LIN {X 0,Y 246.52,Z 385.054,A -85,B 0,C 180,E1 -18943.173,E2 -18943.173} C_VEL
LIN {X 0,Y 246.538,Z 383.912,A -85,B 0,C 180,E1 -18945.451,E2 -18945.451} C_VEL
LIN {X 0,Y 246.771,Z 381.922,A -85,B 0,C 180,E1 -18947.771,E2 -18947.771} C_VEL
LIN {X 0,Y 247.108,Z 378.922,A -85,B 0,C 180,E1 -18950.165,E2 -18950.165} C_VEL
LIN {X 0,Y 247.698,Z 374.789,A -85,B 0,C 180,E1 -18952.602,E2 -18952.602} C_VEL
LIN {X 0,Y 248.557,Z 368.103,A -85,B 0,C 180,E1 -18955.564,E2 -18955.564} C_VEL
LIN {X 0,Y 249.777,Z 360.458,A -85,B 0,C 180,E1 -18958.176,E2 -18958.176} C_VEL
LIN {X 0,Y 250.952,Z 352.88,A -85,B 0,C 180,E1 -18960.245,E2 -18960.245} C_VEL
LIN {X 0,Y 252.424,Z 343.571,A -85,B 0,C 180,E1 -18962.309,E2 -18962.309} C_VEL
LIN {X 0,Y 253.973,Z 333.387,A -85,B 0,C 180,E1 -18964.133,E2 -18964.133} C_VEL
LIN {X 0,Y 255.381,Z 323.073,A -85,B 0,C 180,E1 -18965.62,E2 -18965.62} C_VEL
LIN {X 0,Y 256.697,Z 311.556,A -85,B 0,C 180,E1 -18966.931,E2 -18966.931} C_VEL
LIN {X 0,Y 257.975,Z 298.577,A -85,B 0,C 180,E1 -18968.044,E2 -18968.044} C_VEL
LIN {X 0,Y 258.876,Z 285.337,A -85,B 0,C 180,E1 -18968.84,E2 -18968.84} C_VEL
LIN {X 0,Y 259.602,Z 268.509,A -85,B 0,C 180,E1 -18969.443,E2 -18969.443} C_VEL
LIN {X 0,Y 261.737,Z 209.958,A -85,B 0,C 180,E1 -18971.254,E2 -18971.254} C_VEL
LIN {X 0,Y 260.436,Z 204.838,A -85,B 0,C 180,E1 -18971.54,E2 -18971.54} C_VEL
LIN {X 0,Y 251.175,Z 178.768,A -85,B 0,C 180,E1 -18973.282,E2 -18973.282} C_VEL
LIN {X 0,Y 249.486,Z 174.092,A -85,B 0,C 180,E1 -18973.639,E2 -18973.639} C_VEL
LIN {X 0,Y 249.178,Z 172.45,A -85,B 0,C 180,E1 -18974.354,E2 -18974.354} C_VEL
LIN {X 0,Y 249.215,Z 172.443,A -85,B 0,C 180,E1 -18978.615,E2 -18978.615} C_VEL
LIN {X 0,Y 249.411,Z 172.416,A -85,B 0,C 180,E1 -18981.901,E2 -18981.901} C_VEL
LIN {X 0,Y 249.258,Z 172.435,A -85,B 0,C 180,E1 -18985.148,E2 -18985.148} C_VEL
LIN {X 0,Y 249.654,Z 172.389,A -85,B 0,C 180,E1 -18988.387,E2 -18988.387} C_VEL
LIN {X 0,Y 249.652,Z 172.389,A -85,B 0,C 180,E1 -18991.613,E2 -18991.613} C_VEL
LIN {X 0,Y 249.424,Z 172.416,A -85,B 0,C 180,E1 -18996.472,E2 -18996.472} C_VEL
LIN {X 0,Y 249.33,Z 172.43,A -85,B 0,C 180,E1 -18999.737,E2 -18999.737} C_VEL
LIN {X 0,Y 249.143,Z 172.45,A -85,B 0,C 180,E1 -19004.707,E2 -19004.707} C_VEL
LIN {X 0,Y 249.075,Z 172.459,A -85,B 0,C 180,E1 -19008.082,E2 -19008.082} C_VEL
LIN {X 0,Y 249.039,Z 172.464,A -85,B 0,C 180,E1 -19011.522,E2 -19011.522} C_VEL
LIN {X 0,Y 249.04,Z 172.464,A -85,B 0,C 180,E1 -19015.44,E2 -19015.44} C_VEL
LIN {X 0,Y 249.02,Z 172.465,A -85,B 0,C 180,E1 -19018.968,E2 -19018.968} C_VEL
LIN {X 0,Y 249.022,Z 172.457,A -85,B 0,C 180,E1 -19022.427,E2 -19022.427} C_VEL
LIN {X 0,Y 249.023,Z 172.463,A -85,B 0,C 180,E1 -19026.346,E2 -19026.346} C_VEL
LIN {X 0,Y 248.975,Z 172.467,A -85,B 0,C 180,E1 -19030.484,E2 -19030.484} C_VEL
LIN {X 0,Y 248.958,Z 172.467,A -85,B 0,C 180,E1 -19034.889,E2 -19034.889} C_VEL
LIN {X 0,Y 248.975,Z 172.471,A -85,B 0,C 180,E1 -19037.355,E2 -19037.355} C_VEL
LIN {X 0,Y 249.036,Z 172.461,A -85,B 0,C 180,E1 -19042.202,E2 -19042.202} C_VEL
LIN {X 0,Y 249.039,Z 172.452,A -85,B 0,C 180,E1 -19045.64,E2 -19045.64} C_VEL
LIN {X 0,Y 248.998,Z 172.463,A -85,B 0,C 180,E1 -19049.467,E2 -19049.467} C_VEL
LIN {X 0,Y 249.017,Z 172.465,A -85,B 0,C 180,E1 -19053.157,E2 -19053.157} C_VEL
LIN {X 0,Y 249.002,Z 172.466,A -85,B 0,C 180,E1 -19056.726,E2 -19056.726} C_VEL
LIN {X 0,Y 249.038,Z 172.456,A -85,B 0,C 180,E1 -19060.206,E2 -19060.206} C_VEL
LIN {X 0,Y 249.155,Z 172.44,A -85,B 0,C 180,E1 -19063.617,E2 -19063.617} C_VEL
LIN {X 0,Y 249.214,Z 172.44,A -85,B 0,C 180,E1 -19068.615,E2 -19068.615} C_VEL
LIN {X 0,Y 249.399,Z 172.415,A -85,B 0,C 180,E1 -19071.901,E2 -19071.901} C_VEL
LIN {X 0,Y 249.249,Z 172.424,A -85,B 0,C 180,E1 -19075.148,E2 -19075.148} C_VEL
LIN {X 0,Y 249.651,Z 172.385,A -85,B 0,C 180,E1 -19078.388,E2 -19078.388} C_VEL
LIN {X 0,Y 249.651,Z 172.386,A -85,B 0,C 180,E1 -19081.614,E2 -19081.614} C_VEL
LIN {X 0,Y 249.383,Z 172.411,A -85,B 0,C 180,E1 -19087.292,E2 -19087.292} C_VEL
LIN {X 0,Y 249.329,Z 172.426,A -85,B 0,C 180,E1 -19089.738,E2 -19089.738} C_VEL
LIN {X 0,Y 249.128,Z 172.447,A -85,B 0,C 180,E1 -19094.277,E2 -19094.277} C_VEL
LIN {X 0,Y 248.465,Z 172.533,A -85,B 0,C 180,E1 -19095.626,E2 -19095.626} C_VEL
LIN {X 0,Y 245.549,Z 172.897,A -85,B 0,C 180,E1 -19097.823,E2 -19097.823} C_VEL
LIN {X 0,Y 243.077,Z 173.207,A -85,B 0,C 180,E1 -19099.613,E2 -19099.613} C_VEL
LIN {X 0,Y 242.044,Z 173.334,A -85,B 0,C 180,E1 -19101.004,E2 -19101.004} C_VEL
LIN {X 0,Y 241.976,Z 173.344,A -85,B 0,C 180,E1 -19101.475,E2 -19101.475} C_VEL
LIN {X 0,Y 241.985,Z 173.343,A -85,B 0,C 180,E1 -19105.827,E2 -19105.827} C_VEL
LIN {X 0,Y 241.962,Z 173.345,A -85,B 0,C 180,E1 -19109.59,E2 -19109.59} C_VEL
LIN {X 0,Y 241.978,Z 173.334,A -85,B 0,C 180,E1 -19113.494,E2 -19113.494} C_VEL
LIN {X 0,Y 241.983,Z 173.343,A -85,B 0,C 180,E1 -19117.584,E2 -19117.584} C_VEL
LIN {X 0,Y 241.908,Z 173.351,A -85,B 0,C 180,E1 -19121.93,E2 -19121.93} C_VEL
LIN {X 0,Y 241.901,Z 173.353,A -85,B 0,C 180,E1 -19126.581,E2 -19126.581} C_VEL
LIN {X 0,Y 241.993,Z 173.341,A -85,B 0,C 180,E1 -19131.642,E2 -19131.642} C_VEL
LIN {X 0,Y 242.041,Z 173.508,A -85,B 0,C 180,E1 -19134.69,E2 -19134.69} C_VEL
LIN {X 0,Y 244.216,Z 183.907,A -85,B 0,C 180,E1 -19138.802,E2 -19138.802} C_VEL
LIN {X 0,Y 244.914,Z 187.186,A -85,B 0,C 180,E1 -19139.977,E2 -19139.977} C_VEL
LIN {X 0,Y 250.399,Z 203.541,A -85,B 0,C 180,E1 -19141.083,E2 -19141.083} C_VEL
LIN {X 0,Y 254.531,Z 235.313,A -85,B 0,C 180,E1 -19142.572,E2 -19142.572} C_VEL
LIN {X 0,Y 252.192,Z 295.458,A -85,B 0,C 180,E1 -19144.519,E2 -19144.519} C_VEL
LIN {X 0,Y 251.181,Z 309.454,A -85,B 0,C 180,E1 -19145.295,E2 -19145.295} C_VEL
LIN {X 0,Y 249.963,Z 321.58,A -85,B 0,C 180,E1 -19146.271,E2 -19146.271} C_VEL
LIN {X 0,Y 248.355,Z 333.361,A -85,B 0,C 180,E1 -19147.541,E2 -19147.541} C_VEL
LIN {X 0,Y 246.695,Z 344.807,A -85,B 0,C 180,E1 -19149.139,E2 -19149.139} C_VEL
LIN {X 0,Y 245.152,Z 354.534,A -85,B 0,C 180,E1 -19150.838,E2 -19150.838} C_VEL
LIN {X 0,Y 243.82,Z 363.731,A -85,B 0,C 180,E1 -19152.83,E2 -19152.83} C_VEL
LIN {X 0,Y 242.306,Z 372.873,A -85,B 0,C 180,E1 -19155.298,E2 -19155.298} C_VEL
LIN {X 0,Y 241.13,Z 380.263,A -85,B 0,C 180,E1 -19157.801,E2 -19157.801} C_VEL
LIN {X 0,Y 240.512,Z 385.237,A -85,B 0,C 180,E1 -19159.902,E2 -19159.902} C_VEL
LIN {X 0,Y 240.069,Z 390.04,A -85,B 0,C 180,E1 -19162.43,E2 -19162.43} C_VEL
LIN {X 0,Y 239.841,Z 393.816,A -85,B 0,C 180,E1 -19165.073,E2 -19165.073} C_VEL
LIN {X 0,Y 239.819,Z 395.499,A -85,B 0,C 180,E1 -19166.64,E2 -19166.64} C_VEL
LIN {X 0,Y 239.866,Z 396.856,A -85,B 0,C 180,E1 -19168.321,E2 -19168.321} C_VEL
LIN {X 0,Y 239.915,Z 397.799,A -85,B 0,C 180,E1 -19170,E2 -19170} C_VEL
LIN {X 0,Y 239.832,Z 398.333,A -85,B 0,C 180,E1 -19171.679,E2 -19171.679} C_VEL
LIN {X 0,Y 239.793,Z 398.194,A -85,B 0,C 180,E1 -19174.791,E2 -19174.791} C_VEL
LIN {X 0,Y 239.958,Z 397.405,A -85,B 0,C 180,E1 -19176.727,E2 -19176.727} C_VEL
LIN {X 0,Y 240.237,Z 396.305,A -85,B 0,C 180,E1 -19178.411,E2 -19178.411} C_VEL
LIN {X 0,Y 240.693,Z 394.773,A -85,B 0,C 180,E1 -19180.09,E2 -19180.09} C_VEL
LIN {X 0,Y 241.681,Z 391.683,A -85,B 0,C 180,E1 -19182.597,E2 -19182.597} C_VEL
LIN {X 0,Y 243.041,Z 387.561,A -85,B 0,C 180,E1 -19185.085,E2 -19185.085} C_VEL
LIN {X 0,Y 245.457,Z 381.266,A -85,B 0,C 180,E1 -19187.926,E2 -19187.926} C_VEL
LIN {X 0,Y 247.687,Z 374.209,A -85,B 0,C 180,E1 -19190.434,E2 -19190.434} C_VEL
LIN {X 0,Y 250.436,Z 366.091,A -85,B 0,C 180,E1 -19192.697,E2 -19192.697} C_VEL
LIN {X 0,Y 253.756,Z 355.582,A -85,B 0,C 180,E1 -19194.983,E2 -19194.983} C_VEL
LIN {X 0,Y 256.918,Z 344.741,A -85,B 0,C 180,E1 -19196.83,E2 -19196.83} C_VEL
LIN {X 0,Y 259.555,Z 333.934,A -85,B 0,C 180,E1 -19198.284,E2 -19198.284} C_VEL
LIN {X 0,Y 262.152,Z 322,A -85,B 0,C 180,E1 -19199.512,E2 -19199.512} C_VEL
LIN {X 0,Y 264.304,Z 309.764,A -85,B 0,C 180,E1 -19200.456,E2 -19200.456} C_VEL
LIN {X 0,Y 266.008,Z 296.258,A -85,B 0,C 180,E1 -19201.175,E2 -19201.175} C_VEL
LIN {X 0,Y 267.618,Z 272.839,A -85,B 0,C 180,E1 -19201.955,E2 -19201.955} C_VEL
LIN {X 0,Y 269.551,Z 238.998,A -85,B 0,C 180,E1 -19203.038,E2 -19203.038} C_VEL
LIN {X 0,Y 267.849,Z 225.779,A -85,B 0,C 180,E1 -19203.966,E2 -19203.966} C_VEL
LIN {X 0,Y 263.151,Z 214.762,A -85,B 0,C 180,E1 -19205.482,E2 -19205.482} C_VEL
LIN {X 0,Y 257.726,Z 204.119,A -85,B 0,C 180,E1 -19207.295,E2 -19207.295} C_VEL
LIN {X 0,Y 254.614,Z 198.67,A -85,B 0,C 180,E1 -19208.381,E2 -19208.381} C_VEL
LIN {X 0,Y 251.844,Z 194.026,A -85,B 0,C 180,E1 -19209.398,E2 -19209.398} C_VEL
LIN {X 0,Y 248.589,Z 188.923,A -85,B 0,C 180,E1 -19210.657,E2 -19210.657} C_VEL
LIN {X 0,Y 245.438,Z 184.115,A -85,B 0,C 180,E1 -19211.96,E2 -19211.96} C_VEL
LIN {X 0,Y 245.215,Z 183.565,A -85,B 0,C 180,E1 -19212.132,E2 -19212.132} C_VEL
LIN {X 0,Y 243.265,Z 177.594,A -85,B 0,C 180,E1 -19216.24,E2 -19216.24} C_VEL
LIN {X 0,Y 241.931,Z 173.344,A -85,B 0,C 180,E1 -19219.792,E2 -19219.792} C_VEL
LIN {X 0,Y 241.977,Z 173.34,A -85,B 0,C 180,E1 -19222.415,E2 -19222.415} C_VEL
LIN {X 0,Y 241.976,Z 173.333,A -85,B 0,C 180,E1 -19226.506,E2 -19226.506} C_VEL
LIN {X 0,Y 241.968,Z 173.334,A -85,B 0,C 180,E1 -19230.614,E2 -19230.614} C_VEL
LIN {X 0,Y 241.993,Z 173.331,A -85,B 0,C 180,E1 -19234.196,E2 -19234.196} C_VEL
LIN {X 0,Y 241.982,Z 173.335,A -85,B 0,C 180,E1 -19238.337,E2 -19238.337} C_VEL
LIN {X 0,Y 242.102,Z 173.327,A -85,B 0,C 180,E1 -19243.323,E2 -19243.323} C_VEL
LIN {X 0,Y 242.151,Z 173.312,A -85,B 0,C 180,E1 -19248.277,E2 -19248.277} C_VEL
LIN {X 0,Y 242.363,Z 173.286,A -85,B 0,C 180,E1 -19251.663,E2 -19251.663} C_VEL
LIN {X 0,Y 242.39,Z 173.293,A -85,B 0,C 180,E1 -19253.339,E2 -19253.339} C_VEL
LIN {X 0,Y 242.622,Z 173.362,A -85,B 0,C 180,E1 -19258.651,E2 -19258.651} C_VEL
LIN {X 0,Y 243.758,Z 176.955,A -85,B 0,C 180,E1 -19261.497,E2 -19261.497} C_VEL
LIN {X 0,Y 246.362,Z 181.091,A -85,B 0,C 180,E1 -19262.65,E2 -19262.65} C_VEL
LIN {X 0,Y 251.858,Z 188.789,A -85,B 0,C 180,E1 -19264.801,E2 -19264.801} C_VEL
LIN {X 0,Y 255.288,Z 194.042,A -85,B 0,C 180,E1 -19266.042,E2 -19266.042} C_VEL
LIN {X 0,Y 259.927,Z 201.958,A -85,B 0,C 180,E1 -19267.629,E2 -19267.629} C_VEL
LIN {X 0,Y 264.851,Z 211.136,A -85,B 0,C 180,E1 -19269.21,E2 -19269.21} C_VEL
LIN {X 0,Y 269.644,Z 221.759,A -85,B 0,C 180,E1 -19270.706,E2 -19270.706} C_VEL
LIN {X 0,Y 270.473,Z 224.051,A -85,B 0,C 180,E1 -19270.976,E2 -19270.976} C_VEL
LIN {X 0,Y 266.544,Z 284.682,A -85,B 0,C 180,E1 -19272.905,E2 -19272.905} C_VEL
LIN {X 0,Y 264.995,Z 298.059,A -85,B 0,C 180,E1 -19273.618,E2 -19273.618} C_VEL
LIN {X 0,Y 263.262,Z 309.741,A -85,B 0,C 180,E1 -19274.532,E2 -19274.532} C_VEL
LIN {X 0,Y 260.801,Z 322.218,A -85,B 0,C 180,E1 -19275.833,E2 -19275.833} C_VEL
LIN {X 0,Y 258.191,Z 333.132,A -85,B 0,C 180,E1 -19277.299,E2 -19277.299} C_VEL
LIN {X 0,Y 255.316,Z 343.541,A -85,B 0,C 180,E1 -19279.079,E2 -19279.079} C_VEL
LIN {X 0,Y 252.717,Z 351.897,A -85,B 0,C 180,E1 -19280.856,E2 -19280.856} C_VEL
LIN {X 0,Y 249.787,Z 360.715,A -85,B 0,C 180,E1 -19283.197,E2 -19283.197} C_VEL
LIN {X 0,Y 247.107,Z 368.14,A -85,B 0,C 180,E1 -19285.703,E2 -19285.703} C_VEL
LIN {X 0,Y 244.845,Z 374.061,A -85,B 0,C 180,E1 -19288.305,E2 -19288.305} C_VEL
LIN {X 0,Y 242.789,Z 379.302,A -85,B 0,C 180,E1 -19291.402,E2 -19291.402} C_VEL
LIN {X 0,Y 241.709,Z 381.903,A -85,B 0,C 180,E1 -19293.534,E2 -19293.534} C_VEL
LIN {X 0,Y 240.814,Z 383.848,A -85,B 0,C 180,E1 -19295.709,E2 -19295.709} C_VEL
LIN {X 0,Y 240.184,Z 385.072,A -85,B 0,C 180,E1 -19297.913,E2 -19297.913} C_VEL
LIN {X 0,Y 239.708,Z 385.608,A -85,B 0,C 180,E1 -19300.335,E2 -19300.335} C_VEL
LIN {X 0,Y 239.455,Z 385.3,A -85,B 0,C 180,E1 -19302.8,E2 -19302.8} C_VEL
LIN {X 0,Y 239.441,Z 384.156,A -85,B 0,C 180,E1 -19305.217,E2 -19305.217} C_VEL
LIN {X 0,Y 239.661,Z 382.202,A -85,B 0,C 180,E1 -19307.588,E2 -19307.588} C_VEL
LIN {X 0,Y 239.962,Z 379.445,A -85,B 0,C 180,E1 -19309.885,E2 -19309.885} C_VEL
LIN {X 0,Y 240.617,Z 374.876,A -85,B 0,C 180,E1 -19312.695,E2 -19312.695} C_VEL
LIN {X 0,Y 241.448,Z 368.56,A -85,B 0,C 180,E1 -19315.583,E2 -19315.583} C_VEL
LIN {X 0,Y 242.676,Z 360.955,A -85,B 0,C 180,E1 -19318.284,E2 -19318.284} C_VEL
LIN {X 0,Y 244.076,Z 352.312,A -85,B 0,C 180,E1 -19320.693,E2 -19320.693} C_VEL
LIN {X 0,Y 245.782,Z 341.914,A -85,B 0,C 180,E1 -19323.004,E2 -19323.004} C_VEL
LIN {X 0,Y 247.307,Z 331.92,A -85,B 0,C 180,E1 -19324.77,E2 -19324.77} C_VEL
LIN {X 0,Y 248.952,Z 319.541,A -85,B 0,C 180,E1 -19326.5,E2 -19326.5} C_VEL
LIN {X 0,Y 250.449,Z 307.104,A -85,B 0,C 180,E1 -19327.822,E2 -19327.822} C_VEL
LIN {X 0,Y 251.633,Z 293.248,A -85,B 0,C 180,E1 -19328.899,E2 -19328.899} C_VEL
LIN {X 0,Y 252.49,Z 280.371,A -85,B 0,C 180,E1 -19329.56,E2 -19329.56} C_VEL
LIN {X 0,Y 255.095,Z 211.087,A -85,B 0,C 180,E1 -19331.786,E2 -19331.786} C_VEL
LIN {X 0,Y 253.56,Z 205.589,A -85,B 0,C 180,E1 -19332.112,E2 -19332.112} C_VEL
LIN {X 0,Y 243.979,Z 178.829,A -85,B 0,C 180,E1 -19333.972,E2 -19333.972} C_VEL
LIN {X 0,Y 242.308,Z 174.228,A -85,B 0,C 180,E1 -19334.363,E2 -19334.363} C_VEL
LIN {X 0,Y 242.127,Z 173.329,A -85,B 0,C 180,E1 -19334.857,E2 -19334.857} C_VEL
LIN {X 0,Y 242.309,Z 173.302,A -85,B 0,C 180,E1 -19340.447,E2 -19340.447} C_VEL
LIN {X 0,Y 242.393,Z 173.29,A -85,B 0,C 180,E1 -19343.34,E2 -19343.34} C_VEL
LIN {X 0,Y 242.614,Z 173.266,A -85,B 0,C 180,E1 -19348.34,E2 -19348.34} C_VEL
LIN {X 0,Y 242.611,Z 173.266,A -85,B 0,C 180,E1 -19351.66,E2 -19351.66} C_VEL
LIN {X 0,Y 242.396,Z 173.291,A -85,B 0,C 180,E1 -19356.66,E2 -19356.66} C_VEL
LIN {X 0,Y 242.257,Z 173.311,A -85,B 0,C 180,E1 -19360.024,E2 -19360.024} C_VEL
LIN {X 0,Y 242.101,Z 173.328,A -85,B 0,C 180,E1 -19365.145,E2 -19365.145} C_VEL
LIN {X 0,Y 242.014,Z 173.337,A -85,B 0,C 180,E1 -19368.629,E2 -19368.629} C_VEL
LIN {X 0,Y 241.969,Z 173.343,A -85,B 0,C 180,E1 -19372.184,E2 -19372.184} C_VEL
LIN {X 0,Y 241.983,Z 173.343,A -85,B 0,C 180,E1 -19375.827,E2 -19375.827} C_VEL
LIN {X 0,Y 241.959,Z 173.343,A -85,B 0,C 180,E1 -19379.59,E2 -19379.59} C_VEL
LIN {X 0,Y 241.975,Z 173.341,A -85,B 0,C 180,E1 -19383.493,E2 -19383.493} C_VEL
LIN {X 0,Y 241.98,Z 173.342,A -85,B 0,C 180,E1 -19387.583,E2 -19387.583} C_VEL
LIN {X 0,Y 241.904,Z 173.343,A -85,B 0,C 180,E1 -19391.929,E2 -19391.929} C_VEL
LIN {X 0,Y 241.897,Z 173.349,A -85,B 0,C 180,E1 -19396.58,E2 -19396.58} C_VEL
LIN {X 0,Y 241.989,Z 173.339,A -85,B 0,C 180,E1 -19401.642,E2 -19401.642} C_VEL
LIN {X 0,Y 241.975,Z 173.338,A -85,B 0,C 180,E1 -19404.488,E2 -19404.488} C_VEL
LIN {X 0,Y 241.949,Z 173.337,A -85,B 0,C 180,E1 -19408.477,E2 -19408.477} C_VEL
LIN {X 0,Y 241.957,Z 173.344,A -85,B 0,C 180,E1 -19412.307,E2 -19412.307} C_VEL
LIN {X 0,Y 241.954,Z 173.344,A -85,B 0,C 180,E1 -19416.006,E2 -19416.006} C_VEL
LIN {X 0,Y 241.979,Z 173.333,A -85,B 0,C 180,E1 -19419.604,E2 -19419.604} C_VEL
LIN {X 0,Y 242.103,Z 173.318,A -85,B 0,C 180,E1 -19423.325,E2 -19423.325} C_VEL
LIN {X 0,Y 242.148,Z 173.322,A -85,B 0,C 180,E1 -19428.279,E2 -19428.279} C_VEL
LIN {X 0,Y 242.354,Z 173.291,A -85,B 0,C 180,E1 -19431.664,E2 -19431.664} C_VEL
LIN {X 0,Y 242.387,Z 173.283,A -85,B 0,C 180,E1 -19433.341,E2 -19433.341} C_VEL
LIN {X 0,Y 242.611,Z 173.262,A -85,B 0,C 180,E1 -19438.341,E2 -19438.341} C_VEL
LIN {X 0,Y 242.611,Z 173.263,A -85,B 0,C 180,E1 -19441.661,E2 -19441.661} C_VEL
LIN {X 0,Y 242.387,Z 173.282,A -85,B 0,C 180,E1 -19446.661,E2 -19446.661} C_VEL
LIN {X 0,Y 242.257,Z 173.309,A -85,B 0,C 180,E1 -19450.025,E2 -19450.025} C_VEL
LIN {X 0,Y 242.102,Z 173.325,A -85,B 0,C 180,E1 -19455.146,E2 -19455.146} C_VEL
LIN {X 0,Y 242.014,Z 173.335,A -85,B 0,C 180,E1 -19458.63,E2 -19458.63} C_VEL
LIN {X 0,Y 241.976,Z 173.344,A -85,B 0,C 180,E1 -19461.475,E2 -19461.475} C_VEL
LIN {X 0,Y 241.342,Z 173.429,A -85,B 0,C 180,E1 -19462.865,E2 -19462.865} C_VEL
LIN {X 0,Y 238.476,Z 173.79,A -85,B 0,C 180,E1 -19465.132,E2 -19465.132} C_VEL
LIN {X 0,Y 236.02,Z 174.091,A -85,B 0,C 180,E1 -19466.979,E2 -19466.979} C_VEL
LIN {X 0,Y 234.969,Z 174.217,A -85,B 0,C 180,E1 -19468.413,E2 -19468.413} C_VEL
LIN {X 0,Y 234.887,Z 174.225,A -85,B 0,C 180,E1 -19468.9,E2 -19468.9} C_VEL
LIN {X 0,Y 234.94,Z 174.21,A -85,B 0,C 180,E1 -19473.114,E2 -19473.114} C_VEL
LIN {X 0,Y 234.915,Z 174.221,A -85,B 0,C 180,E1 -19476.752,E2 -19476.752} C_VEL
LIN {X 0,Y 234.912,Z 174.224,A -85,B 0,C 180,E1 -19478.936,E2 -19478.936} C_VEL
LIN {X 0,Y 234.853,Z 174.231,A -85,B 0,C 180,E1 -19483.495,E2 -19483.495} C_VEL
LIN {X 0,Y 234.854,Z 174.23,A -85,B 0,C 180,E1 -19486.507,E2 -19486.507} C_VEL
LIN {X 0,Y 234.919,Z 174.224,A -85,B 0,C 180,E1 -19491.079,E2 -19491.079} C_VEL
LIN {X 0,Y 234.959,Z 174.32,A -85,B 0,C 180,E1 -19494.184,E2 -19494.184} C_VEL
LIN {X 0,Y 237.009,Z 183.957,A -85,B 0,C 180,E1 -19498.126,E2 -19498.126} C_VEL
LIN {X 0,Y 237.581,Z 186.758,A -85,B 0,C 180,E1 -19499.229,E2 -19499.229} C_VEL
LIN {X 0,Y 243.924,Z 205.404,A -85,B 0,C 180,E1 -19500.562,E2 -19500.562} C_VEL
LIN {X 0,Y 247.846,Z 236.255,A -85,B 0,C 180,E1 -19502.044,E2 -19502.044} C_VEL
LIN {X 0,Y 245.475,Z 294.975,A -85,B 0,C 180,E1 -19503.998,E2 -19503.998} C_VEL
LIN {X 0,Y 244.438,Z 309.032,A -85,B 0,C 180,E1 -19504.794,E2 -19504.794} C_VEL
LIN {X 0,Y 243.181,Z 321.203,A -85,B 0,C 180,E1 -19505.794,E2 -19505.794} C_VEL
LIN {X 0,Y 241.523,Z 333.017,A -85,B 0,C 180,E1 -19507.096,E2 -19507.096} C_VEL
LIN {X 0,Y 239.82,Z 344.493,A -85,B 0,C 180,E1 -19508.737,E2 -19508.737} C_VEL
LIN {X 0,Y 238.061,Z 355.267,A -85,B 0,C 180,E1 -19510.688,E2 -19510.688} C_VEL
LIN {X 0,Y 236.713,Z 364.24,A -85,B 0,C 180,E1 -19512.729,E2 -19512.729} C_VEL
LIN {X 0,Y 235.189,Z 373.316,A -85,B 0,C 180,E1 -19515.286,E2 -19515.286} C_VEL
LIN {X 0,Y 233.994,Z 380.569,A -85,B 0,C 180,E1 -19517.863,E2 -19517.863} C_VEL
LIN {X 0,Y 233.293,Z 386.329,A -85,B 0,C 180,E1 -19520.463,E2 -19520.463} C_VEL
LIN {X 0,Y 232.911,Z 390.827,A -85,B 0,C 180,E1 -19523.067,E2 -19523.067} C_VEL
LIN {X 0,Y 232.738,Z 393.693,A -85,B 0,C 180,E1 -19525.215,E2 -19525.215} C_VEL
LIN {X 0,Y 232.778,Z 396.508,A -85,B 0,C 180,E1 -19528.27,E2 -19528.27} C_VEL
LIN {X 0,Y 232.846,Z 397.495,A -85,B 0,C 180,E1 -19530,E2 -19530} C_VEL
LIN {X 0,Y 232.743,Z 398.07,A -85,B 0,C 180,E1 -19531.73,E2 -19531.73} C_VEL
LIN {X 0,Y 232.708,Z 398.096,A -85,B 0,C 180,E1 -19534.697,E2 -19534.697} C_VEL
LIN {X 0,Y 232.896,Z 397.311,A -85,B 0,C 180,E1 -19536.932,E2 -19536.932} C_VEL
LIN {X 0,Y 233.695,Z 394.814,A -85,B 0,C 180,E1 -19540.395,E2 -19540.395} C_VEL
LIN {X 0,Y 234.743,Z 391.807,A -85,B 0,C 180,E1 -19542.976,E2 -19542.976} C_VEL
LIN {X 0,Y 236.197,Z 387.78,A -85,B 0,C 180,E1 -19545.532,E2 -19545.532} C_VEL
LIN {X 0,Y 238.738,Z 381.633,A -85,B 0,C 180,E1 -19548.448,E2 -19548.448} C_VEL
LIN {X 0,Y 241.014,Z 374.852,A -85,B 0,C 180,E1 -19550.977,E2 -19550.977} C_VEL
LIN {X 0,Y 243.956,Z 366.791,A -85,B 0,C 180,E1 -19553.335,E2 -19553.335} C_VEL
LIN {X 0,Y 246.826,Z 358.465,A -85,B 0,C 180,E1 -19555.283,E2 -19555.283} C_VEL
LIN {X 0,Y 250.05,Z 348.301,A -85,B 0,C 180,E1 -19557.175,E2 -19557.175} C_VEL
LIN {X 0,Y 253.098,Z 336.979,A -85,B 0,C 180,E1 -19558.846,E2 -19558.846} C_VEL
LIN {X 0,Y 255.712,Z 325.974,A -85,B 0,C 180,E1 -19560.104,E2 -19560.104} C_VEL
LIN {X 0,Y 258.103,Z 313.824,A -85,B 0,C 180,E1 -19561.154,E2 -19561.154} C_VEL
LIN {X 0,Y 260.18,Z 299.861,A -85,B 0,C 180,E1 -19562.012,E2 -19562.012} C_VEL
LIN {X 0,Y 261.452,Z 286.174,A -85,B 0,C 180,E1 -19562.554,E2 -19562.554} C_VEL
LIN {X 0,Y 264.35,Z 240.388,A -85,B 0,C 180,E1 -19564.031,E2 -19564.031} C_VEL
LIN {X 0,Y 262.962,Z 229.118,A -85,B 0,C 180,E1 -19564.846,E2 -19564.846} C_VEL
LIN {X 0,Y 258.995,Z 219.522,A -85,B 0,C 180,E1 -19566.203,E2 -19566.203} C_VEL
LIN {X 0,Y 253.902,Z 209.137,A -85,B 0,C 180,E1 -19568.017,E2 -19568.017} C_VEL
LIN {X 0,Y 248.898,Z 200.151,A -85,B 0,C 180,E1 -19569.911,E2 -19569.911} C_VEL
LIN {X 0,Y 245.09,Z 194.218,A -85,B 0,C 180,E1 -19571.441,E2 -19571.441} C_VEL
LIN {X 0,Y 241.565,Z 188.827,A -85,B 0,C 180,E1 -19572.994,E2 -19572.994} C_VEL
LIN {X 0,Y 238.175,Z 183.927,A -85,B 0,C 180,E1 -19574.612,E2 -19574.612} C_VEL
LIN {X 0,Y 237.836,Z 183.203,A -85,B 0,C 180,E1 -19574.83,E2 -19574.83} C_VEL
LIN {X 0,Y 236.465,Z 179.185,A -85,B 0,C 180,E1 -19577.989,E2 -19577.989} C_VEL
LIN {X 0,Y 234.913,Z 174.217,A -85,B 0,C 180,E1 -19582.711,E2 -19582.711} C_VEL
LIN {X 0,Y 234.95,Z 174.21,A -85,B 0,C 180,E1 -19587.422,E2 -19587.422} C_VEL
LIN {X 0,Y 234.889,Z 174.222,A -85,B 0,C 180,E1 -19591.397,E2 -19591.397} C_VEL
LIN {X 0,Y 234.911,Z 174.222,A -85,B 0,C 180,E1 -19595.237,E2 -19595.237} C_VEL
LIN {X 0,Y 234.932,Z 174.22,A -85,B 0,C 180,E1 -19598.962,E2 -19598.962} C_VEL
LIN {X 0,Y 235.046,Z 174.207,A -85,B 0,C 180,E1 -19603.097,E2 -19603.097} C_VEL
LIN {X 0,Y 235.083,Z 174.193,A -85,B 0,C 180,E1 -19607.92,E2 -19607.92} C_VEL
LIN {X 0,Y 235.299,Z 174.167,A -85,B 0,C 180,E1 -19611.411,E2 -19611.411} C_VEL
LIN {X 0,Y 235.341,Z 174.168,A -85,B 0,C 180,E1 -19613.139,E2 -19613.139} C_VEL
LIN {X 0,Y 235.229,Z 174.394,A -85,B 0,C 180,E1 -19615.716,E2 -19615.716} C_VEL
LIN {X 0,Y 236.661,Z 177.382,A -85,B 0,C 180,E1 -19618.777,E2 -19618.777} C_VEL
LIN {X 0,Y 239.129,Z 181.058,A -85,B 0,C 180,E1 -19620.052,E2 -19620.052} C_VEL
LIN {X 0,Y 241.056,Z 183.296,A -85,B 0,C 180,E1 -19620.939,E2 -19620.939} C_VEL
LIN {X 0,Y 243.974,Z 187.634,A -85,B 0,C 180,E1 -19622.267,E2 -19622.267} C_VEL
LIN {X 0,Y 248.962,Z 195.02,A -85,B 0,C 180,E1 -19624.3,E2 -19624.3} C_VEL
LIN {X 0,Y 252.953,Z 201.328,A -85,B 0,C 180,E1 -19625.807,E2 -19625.807} C_VEL
LIN {X 0,Y 259.245,Z 212.926,A -85,B 0,C 180,E1 -19628.015,E2 -19628.015} C_VEL
LIN {X 0,Y 264.681,Z 224.885,A -85,B 0,C 180,E1 -19629.813,E2 -19629.813} C_VEL
LIN {X 0,Y 265.189,Z 226.157,A -85,B 0,C 180,E1 -19629.98,E2 -19629.98} C_VEL
LIN {X 0,Y 261.261,Z 284.306,A -85,B 0,C 180,E1 -19631.874,E2 -19631.874} C_VEL
LIN {X 0,Y 259.552,Z 298.137,A -85,B 0,C 180,E1 -19632.609,E2 -19632.609} C_VEL
LIN {X 0,Y 257.583,Z 310.646,A -85,B 0,C 180,E1 -19633.618,E2 -19633.618} C_VEL
LIN {X 0,Y 255.158,Z 322.402,A -85,B 0,C 180,E1 -19634.869,E2 -19634.869} C_VEL
LIN {X 0,Y 252.388,Z 333.377,A -85,B 0,C 180,E1 -19636.36,E2 -19636.36} C_VEL
LIN {X 0,Y 249.649,Z 343.085,A -85,B 0,C 180,E1 -19638.038,E2 -19638.038} C_VEL
LIN {X 0,Y 246.618,Z 352.212,A -85,B 0,C 180,E1 -19639.996,E2 -19639.996} C_VEL
LIN {X 0,Y 243.397,Z 361.316,A -85,B 0,C 180,E1 -19642.487,E2 -19642.487} C_VEL
LIN {X 0,Y 240.524,Z 368.669,A -85,B 0,C 180,E1 -19645.071,E2 -19645.071} C_VEL
LIN {X 0,Y 238.16,Z 374.478,A -85,B 0,C 180,E1 -19647.715,E2 -19647.715} C_VEL
LIN {X 0,Y 236.264,Z 378.948,A -85,B 0,C 180,E1 -19650.387,E2 -19650.387} C_VEL
LIN {X 0,Y 234.803,Z 382.209,A -85,B 0,C 180,E1 -19653.064,E2 -19653.064} C_VEL
LIN {X 0,Y 233.7,Z 384.375,A -85,B 0,C 180,E1 -19655.713,E2 -19655.713} C_VEL
LIN {X 0,Y 232.99,Z 385.553,A -85,B 0,C 180,E1 -19658.348,E2 -19658.348} C_VEL
LIN {X 0,Y 232.416,Z 385.714,A -85,B 0,C 180,E1 -19661.701,E2 -19661.701} C_VEL
LIN {X 0,Y 232.332,Z 384.885,A -85,B 0,C 180,E1 -19664.086,E2 -19664.086} C_VEL
LIN {X 0,Y 232.428,Z 383.245,A -85,B 0,C 180,E1 -19666.526,E2 -19666.526} C_VEL
LIN {X 0,Y 232.734,Z 380.69,A -85,B 0,C 180,E1 -19669.019,E2 -19669.019} C_VEL
LIN {X 0,Y 233.416,Z 375.824,A -85,B 0,C 180,E1 -19672.303,E2 -19672.303} C_VEL
LIN {X 0,Y 234.199,Z 369.876,A -85,B 0,C 180,E1 -19675.239,E2 -19675.239} C_VEL
LIN {X 0,Y 235.383,Z 362.595,A -85,B 0,C 180,E1 -19677.997,E2 -19677.997} C_VEL
LIN {X 0,Y 236.586,Z 355.499,A -85,B 0,C 180,E1 -19680.161,E2 -19680.161} C_VEL
LIN {X 0,Y 238.04,Z 346.775,A -85,B 0,C 180,E1 -19682.34,E2 -19682.34} C_VEL
LIN {X 0,Y 239.537,Z 337.711,A -85,B 0,C 180,E1 -19684.184,E2 -19684.184} C_VEL
LIN {X 0,Y 241.133,Z 327.138,A -85,B 0,C 180,E1 -19685.919,E2 -19685.919} C_VEL
LIN {X 0,Y 242.719,Z 314.927,A -85,B 0,C 180,E1 -19687.497,E2 -19687.497} C_VEL
LIN {X 0,Y 244.117,Z 302.802,A -85,B 0,C 180,E1 -19688.687,E2 -19688.687} C_VEL
LIN {X 0,Y 245.217,Z 288.818,A -85,B 0,C 180,E1 -19689.666,E2 -19689.666} C_VEL
LIN {X 0,Y 245.974,Z 275.964,A -85,B 0,C 180,E1 -19690.237,E2 -19690.237} C_VEL
LIN {X 0,Y 248.432,Z 211.688,A -85,B 0,C 180,E1 -19692.345,E2 -19692.345} C_VEL
LIN {X 0,Y 238.972,Z 184.652,A -85,B 0,C 180,E1 -19694.256,E2 -19694.256} C_VEL
LIN {X 0,Y 235.126,Z 174.52,A -85,B 0,C 180,E1 -19695.061,E2 -19695.061} C_VEL
LIN {X 0,Y 235.071,Z 174.208,A -85,B 0,C 180,E1 -19695.279,E2 -19695.279} C_VEL
LIN {X 0,Y 235.262,Z 174.181,A -85,B 0,C 180,E1 -19700.331,E2 -19700.331} C_VEL
LIN {X 0,Y 235.344,Z 174.168,A -85,B 0,C 180,E1 -19703.14,E2 -19703.14} C_VEL
LIN {X 0,Y 235.573,Z 174.144,A -85,B 0,C 180,E1 -19708.291,E2 -19708.291} C_VEL
LIN {X 0,Y 235.57,Z 174.144,A -85,B 0,C 180,E1 -19711.71,E2 -19711.71} C_VEL
LIN {X 0,Y 235.348,Z 174.169,A -85,B 0,C 180,E1 -19716.86,E2 -19716.86} C_VEL
LIN {X 0,Y 235.181,Z 174.191,A -85,B 0,C 180,E1 -19720.329,E2 -19720.329} C_VEL
LIN {X 0,Y 235.054,Z 174.208,A -85,B 0,C 180,E1 -19725.611,E2 -19725.611} C_VEL
LIN {X 0,Y 234.955,Z 174.218,A -85,B 0,C 180,E1 -19729.21,E2 -19729.21} C_VEL
LIN {X 0,Y 234.905,Z 174.223,A -85,B 0,C 180,E1 -19732.889,E2 -19732.889} C_VEL
LIN {X 0,Y 234.919,Z 174.221,A -85,B 0,C 180,E1 -19736.663,E2 -19736.663} C_VEL
LIN {X 0,Y 234.891,Z 174.22,A -85,B 0,C 180,E1 -19740.573,E2 -19740.573} C_VEL
LIN {X 0,Y 234.922,Z 174.218,A -85,B 0,C 180,E1 -19744.639,E2 -19744.639} C_VEL
LIN {X 0,Y 234.908,Z 174.224,A -85,B 0,C 180,E1 -19748.935,E2 -19748.935} C_VEL
LIN {X 0,Y 234.849,Z 174.222,A -85,B 0,C 180,E1 -19753.494,E2 -19753.494} C_VEL
LIN {X 0,Y 234.849,Z 174.226,A -85,B 0,C 180,E1 -19756.506,E2 -19756.506} C_VEL
LIN {X 0,Y 234.914,Z 174.223,A -85,B 0,C 180,E1 -19761.079,E2 -19761.079} C_VEL
LIN {X 0,Y 234.922,Z 174.21,A -85,B 0,C 180,E1 -19765.361,E2 -19765.361} C_VEL
LIN {X 0,Y 234.895,Z 174.219,A -85,B 0,C 180,E1 -19769.428,E2 -19769.428} C_VEL
LIN {X 0,Y 234.937,Z 174.218,A -85,B 0,C 180,E1 -19773.821,E2 -19773.821} C_VEL
LIN {X 0,Y 234.932,Z 174.212,A -85,B 0,C 180,E1 -19778.963,E2 -19778.963} C_VEL
LIN {X 0,Y 235.046,Z 174.196,A -85,B 0,C 180,E1 -19783.098,E2 -19783.098} C_VEL
LIN {X 0,Y 235.08,Z 174.2,A -85,B 0,C 180,E1 -19787.921,E2 -19787.921} C_VEL
LIN {X 0,Y 235.293,Z 174.17,A -85,B 0,C 180,E1 -19791.412,E2 -19791.412} C_VEL
LIN {X 0,Y 235.337,Z 174.161,A -85,B 0,C 180,E1 -19793.14,E2 -19793.14} C_VEL
LIN {X 0,Y 235.57,Z 174.139,A -85,B 0,C 180,E1 -19798.291,E2 -19798.291} C_VEL
LIN {X 0,Y 235.57,Z 174.14,A -85,B 0,C 180,E1 -19801.71,E2 -19801.71} C_VEL
LIN {X 0,Y 235.338,Z 174.159,A -85,B 0,C 180,E1 -19806.861,E2 -19806.861} C_VEL
LIN {X 0,Y 235.182,Z 174.188,A -85,B 0,C 180,E1 -19810.33,E2 -19810.33} C_VEL
LIN {X 0,Y 235.055,Z 174.202,A -85,B 0,C 180,E1 -19815.611,E2 -19815.611} C_VEL
LIN {X 0,Y 234.956,Z 174.216,A -85,B 0,C 180,E1 -19819.211,E2 -19819.211} C_VEL
LIN {X 0,Y 234.906,Z 174.222,A -85,B 0,C 180,E1 -19822.889,E2 -19822.889} C_VEL
LIN {X 0,Y 234.904,Z 174.224,A -85,B 0,C 180,E1 -19826.666,E2 -19826.666} C_VEL
LIN {X 0,Y 234.887,Z 174.225,A -85,B 0,C 180,E1 -19828.9,E2 -19828.9} C_VEL
LIN {X 0,Y 234.221,Z 174.308,A -85,B 0,C 180,E1 -19830.332,E2 -19830.332} C_VEL
LIN {X 0,Y 231.359,Z 174.659,A -85,B 0,C 180,E1 -19832.668,E2 -19832.668} C_VEL
LIN {X 0,Y 228.944,Z 174.96,A -85,B 0,C 180,E1 -19834.573,E2 -19834.573} C_VEL
LIN {X 0,Y 227.939,Z 175.089,A -85,B 0,C 180,E1 -19836.052,E2 -19836.052} C_VEL
LIN {X 0,Y 227.874,Z 175.097,A -85,B 0,C 180,E1 -19836.553,E2 -19836.553} C_VEL
LIN {X 0,Y 227.801,Z 175.107,A -85,B 0,C 180,E1 -19840.383,E2 -19840.383} C_VEL
LIN {X 0,Y 227.811,Z 175.109,A -85,B 0,C 180,E1 -19845.2,E2 -19845.2} C_VEL
LIN {X 0,Y 227.801,Z 175.109,A -85,B 0,C 180,E1 -19849.618,E2 -19849.618} C_VEL
LIN {X 0,Y 227.929,Z 175.279,A -85,B 0,C 180,E1 -19853.726,E2 -19853.726} C_VEL
LIN {X 0,Y 230.27,Z 186.291,A -85,B 0,C 180,E1 -19858.361,E2 -19858.361} C_VEL
LIN {X 0,Y 230.42,Z 186.92,A -85,B 0,C 180,E1 -19858.488,E2 -19858.488} C_VEL
LIN {X 0,Y 237.481,Z 207.298,A -85,B 0,C 180,E1 -19860.013,E2 -19860.013} C_VEL
LIN {X 0,Y 241.184,Z 236.477,A -85,B 0,C 180,E1 -19861.468,E2 -19861.468} C_VEL
LIN {X 0,Y 238.78,Z 294.396,A -85,B 0,C 180,E1 -19863.448,E2 -19863.448} C_VEL
LIN {X 0,Y 237.77,Z 307.836,A -85,B 0,C 180,E1 -19864.211,E2 -19864.211} C_VEL
LIN {X 0,Y 236.418,Z 320.806,A -85,B 0,C 180,E1 -19865.289,E2 -19865.289} C_VEL
LIN {X 0,Y 234.707,Z 332.674,A -85,B 0,C 180,E1 -19866.625,E2 -19866.625} C_VEL
LIN {X 0,Y 232.957,Z 344.178,A -85,B 0,C 180,E1 -19868.311,E2 -19868.311} C_VEL
LIN {X 0,Y 231.188,Z 354.59,A -85,B 0,C 180,E1 -19870.233,E2 -19870.233} C_VEL
LIN {X 0,Y 229.884,Z 363.142,A -85,B 0,C 180,E1 -19872.199,E2 -19872.199} C_VEL
LIN {X 0,Y 228.269,Z 372.37,A -85,B 0,C 180,E1 -19874.829,E2 -19874.829} C_VEL
LIN {X 0,Y 227.005,Z 379.783,A -85,B 0,C 180,E1 -19877.484,E2 -19877.484} C_VEL
LIN {X 0,Y 226.263,Z 385.689,A -85,B 0,C 180,E1 -19880.163,E2 -19880.163} C_VEL
LIN {X 0,Y 225.836,Z 390.292,A -85,B 0,C 180,E1 -19882.849,E2 -19882.849} C_VEL
LIN {X 0,Y 225.641,Z 393.553,A -85,B 0,C 180,E1 -19885.353,E2 -19885.353} C_VEL
LIN {X 0,Y 225.691,Z 396.157,A -85,B 0,C 180,E1 -19888.215,E2 -19888.215} C_VEL
LIN {X 0,Y 225.779,Z 397.188,A -85,B 0,C 180,E1 -19890,E2 -19890} C_VEL
LIN {X 0,Y 225.657,Z 397.803,A -85,B 0,C 180,E1 -19891.784,E2 -19891.784} C_VEL
LIN {X 0,Y 225.599,Z 397.96,A -85,B 0,C 180,E1 -19894.515,E2 -19894.515} C_VEL
LIN {X 0,Y 225.828,Z 397.229,A -85,B 0,C 180,E1 -19897.151,E2 -19897.151} C_VEL
LIN {X 0,Y 226.682,Z 394.827,A -85,B 0,C 180,E1 -19900.72,E2 -19900.72} C_VEL
LIN {X 0,Y 227.793,Z 391.915,A -85,B 0,C 180,E1 -19903.379,E2 -19903.379} C_VEL
LIN {X 0,Y 229.373,Z 387.994,A -85,B 0,C 180,E1 -19906.007,E2 -19906.007} C_VEL
LIN {X 0,Y 231.597,Z 382.979,A -85,B 0,C 180,E1 -19908.58,E2 -19908.58} C_VEL
LIN {X 0,Y 233.939,Z 376.74,A -85,B 0,C 180,E1 -19911.131,E2 -19911.131} C_VEL
LIN {X 0,Y 236.916,Z 369.011,A -85,B 0,C 180,E1 -19913.607,E2 -19913.607} C_VEL
LIN {X 0,Y 240.472,Z 359.372,A -85,B 0,C 180,E1 -19916,E2 -19916} C_VEL
LIN {X 0,Y 243.84,Z 349.493,A -85,B 0,C 180,E1 -19917.927,E2 -19917.927} C_VEL
LIN {X 0,Y 247.013,Z 338.577,A -85,B 0,C 180,E1 -19919.626,E2 -19919.626} C_VEL
LIN {X 0,Y 249.702,Z 328.056,A -85,B 0,C 180,E1 -19920.907,E2 -19920.907} C_VEL
LIN {X 0,Y 252.379,Z 315.626,A -85,B 0,C 180,E1 -19922.061,E2 -19922.061} C_VEL
LIN {X 0,Y 254.554,Z 302.597,A -85,B 0,C 180,E1 -19922.925,E2 -19922.925} C_VEL
LIN {X 0,Y 256.086,Z 288.653,A -85,B 0,C 180,E1 -19923.534,E2 -19923.534} C_VEL
LIN {X 0,Y 259.223,Z 241.577,A -85,B 0,C 180,E1 -19925.078,E2 -19925.078} C_VEL
LIN {X 0,Y 258.08,Z 232.128,A -85,B 0,C 180,E1 -19925.794,E2 -19925.794} C_VEL
LIN {X 0,Y 254.072,Z 222.344,A -85,B 0,C 180,E1 -19927.277,E2 -19927.277} C_VEL
LIN {X 0,Y 248.937,Z 211.941,A -85,B 0,C 180,E1 -19929.226,E2 -19929.226} C_VEL
LIN {X 0,Y 244.935,Z 204.771,A -85,B 0,C 180,E1 -19930.853,E2 -19930.853} C_VEL
LIN {X 0,Y 241.68,Z 199.491,A -85,B 0,C 180,E1 -19932.251,E2 -19932.251} C_VEL
LIN {X 0,Y 238.667,Z 194.687,A -85,B 0,C 180,E1 -19933.665,E2 -19933.665} C_VEL
LIN {X 0,Y 235.214,Z 189.474,A -85,B 0,C 180,E1 -19935.408,E2 -19935.408} C_VEL
LIN {X 0,Y 230.831,Z 183.601,A -85,B 0,C 180,E1 -19937.874,E2 -19937.874} C_VEL
LIN {X 0,Y 230.345,Z 182.631,A -85,B 0,C 180,E1 -19938.278,E2 -19938.278} C_VEL
LIN {X 0,Y 228.799,Z 177.829,A -85,B 0,C 180,E1 -19942.999,E2 -19942.999} C_VEL
LIN {X 0,Y 227.875,Z 175.089,A -85,B 0,C 180,E1 -19946.532,E2 -19946.532} C_VEL
LIN {X 0,Y 227.869,Z 175.089,A -85,B 0,C 180,E1 -19950.43,E2 -19950.43} C_VEL
LIN {X 0,Y 227.868,Z 175.091,A -85,B 0,C 180,E1 -19954.418,E2 -19954.418} C_VEL
LIN {X 0,Y 227.915,Z 175.086,A -85,B 0,C 180,E1 -19958.282,E2 -19958.282} C_VEL
LIN {X 0,Y 227.996,Z 175.077,A -85,B 0,C 180,E1 -19963.893,E2 -19963.893} C_VEL
LIN {X 0,Y 228.122,Z 175.063,A -85,B 0,C 180,E1 -19969.347,E2 -19969.347} C_VEL
LIN {X 0,Y 228.265,Z 175.121,A -85,B 0,C 180,E1 -19971.813,E2 -19971.813} C_VEL
LIN {X 0,Y 229.296,Z 178.121,A -85,B 0,C 180,E1 -19975.329,E2 -19975.329} C_VEL
LIN {X 0,Y 231.872,Z 181.627,A -85,B 0,C 180,E1 -19976.954,E2 -19976.954} C_VEL
LIN {X 0,Y 234.235,Z 183.846,A -85,B 0,C 180,E1 -19978.221,E2 -19978.221} C_VEL
LIN {X 0,Y 237.312,Z 188.051,A -85,B 0,C 180,E1 -19979.84,E2 -19979.84} C_VEL
LIN {X 0,Y 238.461,Z 189.745,A -85,B 0,C 180,E1 -19980.408,E2 -19980.408} C_VEL
LIN {X 0,Y 245.176,Z 199.786,A -85,B 0,C 180,E1 -19983.414,E2 -19983.414} C_VEL
LIN {X 0,Y 249.269,Z 206.425,A -85,B 0,C 180,E1 -19985.047,E2 -19985.047} C_VEL
LIN {X 0,Y 255.176,Z 217.654,A -85,B 0,C 180,E1 -19987.248,E2 -19987.248} C_VEL
LIN {X 0,Y 259.974,Z 228.433,A -85,B 0,C 180,E1 -19988.953,E2 -19988.953} C_VEL
LIN {X 0,Y 256.011,Z 284.715,A -85,B 0,C 180,E1 -19990.818,E2 -19990.818} C_VEL
LIN {X 0,Y 254.249,Z 298.448,A -85,B 0,C 180,E1 -19991.56,E2 -19991.56} C_VEL
LIN {X 0,Y 252.278,Z 310.501,A -85,B 0,C 180,E1 -19992.54,E2 -19992.54} C_VEL
LIN {X 0,Y 249.657,Z 322.578,A -85,B 0,C 180,E1 -19993.843,E2 -19993.843} C_VEL
LIN {X 0,Y 246.873,Z 333.08,A -85,B 0,C 180,E1 -19995.29,E2 -19995.29} C_VEL
LIN {X 0,Y 243.796,Z 343.333,A -85,B 0,C 180,E1 -19997.085,E2 -19997.085} C_VEL
LIN {X 0,Y 240.69,Z 352.233,A -85,B 0,C 180,E1 -19999.02,E2 -19999.02} C_VEL
LIN {X 0,Y 237.753,Z 360.163,A -85,B 0,C 180,E1 -20001.186,E2 -20001.186} C_VEL
LIN {X 0,Y 234.585,Z 367.915,A -85,B 0,C 180,E1 -20003.856,E2 -20003.856} C_VEL
LIN {X 0,Y 232.375,Z 373,A -85,B 0,C 180,E1 -20006.092,E2 -20006.092} C_VEL
LIN {X 0,Y 229.85,Z 378.564,A -85,B 0,C 180,E1 -20009.289,E2 -20009.289} C_VEL
LIN {X 0,Y 228.48,Z 381.445,A -85,B 0,C 180,E1 -20011.527,E2 -20011.527} C_VEL
LIN {X 0,Y 227.333,Z 383.612,A -85,B 0,C 180,E1 -20013.811,E2 -20013.811} C_VEL
LIN {X 0,Y 226.428,Z 385.141,A -85,B 0,C 180,E1 -20016.198,E2 -20016.198} C_VEL
LIN {X 0,Y 225.766,Z 385.978,A -85,B 0,C 180,E1 -20018.902,E2 -20018.902} C_VEL
LIN {X 0,Y 225.333,Z 385.899,A -85,B 0,C 180,E1 -20021.537,E2 -20021.537} C_VEL
LIN {X 0,Y 225.231,Z 384.942,A -85,B 0,C 180,E1 -20024.138,E2 -20024.138} C_VEL
LIN {X 0,Y 225.337,Z 383.175,A -85,B 0,C 180,E1 -20026.675,E2 -20026.675} C_VEL
LIN {X 0,Y 225.648,Z 380.618,A -85,B 0,C 180,E1 -20029.153,E2 -20029.153} C_VEL
LIN {X 0,Y 226.11,Z 377.28,A -85,B 0,C 180,E1 -20031.565,E2 -20031.565} C_VEL
LIN {X 0,Y 226.87,Z 371.92,A -85,B 0,C 180,E1 -20034.491,E2 -20034.491} C_VEL
LIN {X 0,Y 227.976,Z 364.807,A -85,B 0,C 180,E1 -20037.482,E2 -20037.482} C_VEL
LIN {X 0,Y 229.429,Z 356.549,A -85,B 0,C 180,E1 -20040.176,E2 -20040.176} C_VEL
LIN {X 0,Y 230.959,Z 347.74,A -85,B 0,C 180,E1 -20042.48,E2 -20042.48} C_VEL
LIN {X 0,Y 232.514,Z 338.438,A -85,B 0,C 180,E1 -20044.456,E2 -20044.456} C_VEL
LIN {X 0,Y 234.266,Z 327.324,A -85,B 0,C 180,E1 -20046.344,E2 -20046.344} C_VEL
LIN {X 0,Y 236,Z 314.519,A -85,B 0,C 180,E1 -20048.034,E2 -20048.034} C_VEL
LIN {X 0,Y 237.429,Z 301.973,A -85,B 0,C 180,E1 -20049.27,E2 -20049.27} C_VEL
LIN {X 0,Y 238.496,Z 288.944,A -85,B 0,C 180,E1 -20050.194,E2 -20050.194} C_VEL
LIN {X 0,Y 239.264,Z 276.16,A -85,B 0,C 180,E1 -20050.777,E2 -20050.777} C_VEL
LIN {X 0,Y 241.864,Z 213.418,A -85,B 0,C 180,E1 -20052.882,E2 -20052.882} C_VEL
LIN {X 0,Y 232.835,Z 187.449,A -85,B 0,C 180,E1 -20054.778,E2 -20054.778} C_VEL
LIN {X 0,Y 228.172,Z 175.863,A -85,B 0,C 180,E1 -20055.735,E2 -20055.735} C_VEL
LIN {X 0,Y 228.035,Z 175.085,A -85,B 0,C 180,E1 -20055.84,E2 -20055.84} C_VEL
LIN {X 0,Y 228.236,Z 175.051,A -85,B 0,C 180,E1 -20061.144,E2 -20061.144} C_VEL
LIN {X 0,Y 228.295,Z 175.047,A -85,B 0,C 180,E1 -20062.927,E2 -20062.927} C_VEL
LIN {X 0,Y 228.531,Z 175.022,A -85,B 0,C 180,E1 -20068.238,E2 -20068.238} C_VEL
LIN {X 0,Y 228.529,Z 175.022,A -85,B 0,C 180,E1 -20071.763,E2 -20071.763} C_VEL
LIN {X 0,Y 228.301,Z 175.047,A -85,B 0,C 180,E1 -20077.073,E2 -20077.073} C_VEL
LIN {X 0,Y 228.122,Z 175.069,A -85,B 0,C 180,E1 -20080.652,E2 -20080.652} C_VEL
LIN {X 0,Y 228.005,Z 175.083,A -85,B 0,C 180,E1 -20086.106,E2 -20086.106} C_VEL
LIN {X 0,Y 227.916,Z 175.096,A -85,B 0,C 180,E1 -20091.718,E2 -20091.718} C_VEL
LIN {X 0,Y 227.898,Z 175.095,A -85,B 0,C 180,E1 -20096.581,E2 -20096.581} C_VEL
LIN {X 0,Y 227.866,Z 175.095,A -85,B 0,C 180,E1 -20100.279,E2 -20100.279} C_VEL
LIN {X 0,Y 227.873,Z 175.097,A -85,B 0,C 180,E1 -20103.721,E2 -20103.721} C_VEL
LIN {X 0,Y 227.837,Z 175.102,A -85,B 0,C 180,E1 -20108.092,E2 -20108.092} C_VEL
LIN {X 0,Y 227.782,Z 175.102,A -85,B 0,C 180,E1 -20112.749,E2 -20112.749} C_VEL
LIN {X 0,Y 227.782,Z 175.111,A -85,B 0,C 180,E1 -20117.252,E2 -20117.252} C_VEL
LIN {X 0,Y 227.836,Z 175.101,A -85,B 0,C 180,E1 -20121.908,E2 -20121.908} C_VEL
LIN {X 0,Y 227.875,Z 175.087,A -85,B 0,C 180,E1 -20126.378,E2 -20126.378} C_VEL
LIN {X 0,Y 227.872,Z 175.095,A -85,B 0,C 180,E1 -20130.432,E2 -20130.432} C_VEL
LIN {X 0,Y 227.863,Z 175.102,A -85,B 0,C 180,E1 -20134.419,E2 -20134.419} C_VEL
LIN {X 0,Y 227.915,Z 175.091,A -85,B 0,C 180,E1 -20138.283,E2 -20138.283} C_VEL
LIN {X 0,Y 227.996,Z 175.075,A -85,B 0,C 180,E1 -20143.894,E2 -20143.894} C_VEL
LIN {X 0,Y 228.122,Z 175.065,A -85,B 0,C 180,E1 -20149.348,E2 -20149.348} C_VEL
LIN {X 0,Y 228.289,Z 175.038,A -85,B 0,C 180,E1 -20152.927,E2 -20152.927} C_VEL
LIN {X 0,Y 228.528,Z 175.015,A -85,B 0,C 180,E1 -20158.238,E2 -20158.238} C_VEL
LIN {X 0,Y 228.528,Z 175.018,A -85,B 0,C 180,E1 -20161.763,E2 -20161.763} C_VEL
LIN {X 0,Y 228.29,Z 175.036,A -85,B 0,C 180,E1 -20167.074,E2 -20167.074} C_VEL
LIN {X 0,Y 228.123,Z 175.067,A -85,B 0,C 180,E1 -20170.653,E2 -20170.653} C_VEL
LIN {X 0,Y 228.006,Z 175.076,A -85,B 0,C 180,E1 -20176.107,E2 -20176.107} C_VEL
LIN {X 0,Y 227.917,Z 175.096,A -85,B 0,C 180,E1 -20181.718,E2 -20181.718} C_VEL
LIN {X 0,Y 227.869,Z 175.1,A -85,B 0,C 180,E1 -20186.566,E2 -20186.566} C_VEL
LIN {X 0,Y 227.869,Z 175.098,A -85,B 0,C 180,E1 -20190.279,E2 -20190.279} C_VEL
LIN {X 0,Y 227.876,Z 175.088,A -85,B 0,C 180,E1 -20193.721,E2 -20193.721} C_VEL
LIN {X 0,Y 227.874,Z 175.097,A -85,B 0,C 180,E1 -20196.553,E2 -20196.553} C_VEL
LIN {X 0,Y 227.579,Z 175.137,A -85,B 0,C 180,E1 -20197.539,E2 -20197.539} C_VEL
LIN {X 0,Y 226.221,Z 175.307,A -85,B 0,C 180,E1 -20198.995,E2 -20198.995} C_VEL
LIN {X 0,Y 221.829,Z 175.853,A -85,B 0,C 180,E1 -20202.393,E2 -20202.393} C_VEL
LIN {X 0,Y 220.81,Z 175.98,A -85,B 0,C 180,E1 -20203.919,E2 -20203.919} C_VEL
LIN {X 0,Y 220.752,Z 175.987,A -85,B 0,C 180,E1 -20204.436,E2 -20204.436} C_VEL
LIN {X 0,Y 220.749,Z 175.987,A -85,B 0,C 180,E1 -20208.043,E2 -20208.043} C_VEL
LIN {X 0,Y 220.827,Z 175.98,A -85,B 0,C 180,E1 -20212.794,E2 -20212.794} C_VEL
LIN {X 0,Y 220.896,Z 176.206,A -85,B 0,C 180,E1 -20213.235,E2 -20213.235} C_VEL
LIN {X 0,Y 223.119,Z 186.612,A -85,B 0,C 180,E1 -20217.674,E2 -20217.674} C_VEL
LIN {X 0,Y 230.966,Z 209.015,A -85,B 0,C 180,E1 -20219.424,E2 -20219.424} C_VEL
LIN {X 0,Y 234.533,Z 237.265,A -85,B 0,C 180,E1 -20220.881,E2 -20220.881} C_VEL
LIN {X 0,Y 232.027,Z 294.899,A -85,B 0,C 180,E1 -20222.917,E2 -20222.917} C_VEL
LIN {X 0,Y 230.926,Z 308.829,A -85,B 0,C 180,E1 -20223.753,E2 -20223.753} C_VEL
LIN {X 0,Y 229.546,Z 321.461,A -85,B 0,C 180,E1 -20224.861,E2 -20224.861} C_VEL
LIN {X 0,Y 227.631,Z 333.889,A -85,B 0,C 180,E1 -20226.336,E2 -20226.336} C_VEL
LIN {X 0,Y 226.108,Z 343.846,A -85,B 0,C 180,E1 -20227.86,E2 -20227.86} C_VEL
LIN {X 0,Y 224.275,Z 354.275,A -85,B 0,C 180,E1 -20229.836,E2 -20229.836} C_VEL
LIN {X 0,Y 223.006,Z 361.944,A -85,B 0,C 180,E1 -20231.63,E2 -20231.63} C_VEL
LIN {X 0,Y 221.626,Z 369.993,A -85,B 0,C 180,E1 -20233.891,E2 -20233.891} C_VEL
LIN {X 0,Y 220.219,Z 377.797,A -85,B 0,C 180,E1 -20236.622,E2 -20236.622} C_VEL
LIN {X 0,Y 219.482,Z 383.129,A -85,B 0,C 180,E1 -20238.923,E2 -20238.923} C_VEL
LIN {X 0,Y 218.902,Z 388.255,A -85,B 0,C 180,E1 -20241.693,E2 -20241.693} C_VEL
LIN {X 0,Y 218.633,Z 392.184,A -85,B 0,C 180,E1 -20244.466,E2 -20244.466} C_VEL
LIN {X 0,Y 218.54,Z 394.184,A -85,B 0,C 180,E1 -20246.312,E2 -20246.312} C_VEL
LIN {X 0,Y 218.606,Z 395.755,A -85,B 0,C 180,E1 -20248.157,E2 -20248.157} C_VEL
LIN {X 0,Y 218.689,Z 396.869,A -85,B 0,C 180,E1 -20250,E2 -20250} C_VEL
LIN {X 0,Y 218.572,Z 397.532,A -85,B 0,C 180,E1 -20251.842,E2 -20251.842} C_VEL
LIN {X 0,Y 218.571,Z 397.679,A -85,B 0,C 180,E1 -20255.535,E2 -20255.535} C_VEL
LIN {X 0,Y 218.767,Z 397.147,A -85,B 0,C 180,E1 -20257.383,E2 -20257.383} C_VEL
LIN {X 0,Y 219.689,Z 394.843,A -85,B 0,C 180,E1 -20261.066,E2 -20261.066} C_VEL
LIN {X 0,Y 220.864,Z 392.049,A -85,B 0,C 180,E1 -20263.807,E2 -20263.807} C_VEL
LIN {X 0,Y 222.569,Z 388.255,A -85,B 0,C 180,E1 -20266.51,E2 -20266.51} C_VEL
LIN {X 0,Y 224.902,Z 383.359,A -85,B 0,C 180,E1 -20269.154,E2 -20269.154} C_VEL
LIN {X 0,Y 227.348,Z 377.25,A -85,B 0,C 180,E1 -20271.774,E2 -20271.774} C_VEL
LIN {X 0,Y 230.484,Z 369.695,A -85,B 0,C 180,E1 -20274.308,E2 -20274.308} C_VEL
LIN {X 0,Y 233.462,Z 362.08,A -85,B 0,C 180,E1 -20276.36,E2 -20276.36} C_VEL
LIN {X 0,Y 237.344,Z 351.813,A -85,B 0,C 180,E1 -20278.52,E2 -20278.52} C_VEL
LIN {X 0,Y 240.595,Z 341.508,A -85,B 0,C 180,E1 -20280.257,E2 -20280.257} C_VEL
LIN {X 0,Y 243.74,Z 330.186,A -85,B 0,C 180,E1 -20281.75,E2 -20281.75} C_VEL
LIN {X 0,Y 246.744,Z 317.326,A -85,B 0,C 180,E1 -20283.006,E2 -20283.006} C_VEL
LIN {X 0,Y 249.205,Z 303.675,A -85,B 0,C 180,E1 -20283.968,E2 -20283.968} C_VEL
LIN {X 0,Y 250.764,Z 291.095,A -85,B 0,C 180,E1 -20284.553,E2 -20284.553} C_VEL
LIN {X 0,Y 254.209,Z 242.518,A -85,B 0,C 180,E1 -20286.203,E2 -20286.203} C_VEL
LIN {X 0,Y 253.369,Z 235.242,A -85,B 0,C 180,E1 -20286.783,E2 -20286.783} C_VEL
LIN {X 0,Y 249.61,Z 226.049,A -85,B 0,C 180,E1 -20288.246,E2 -20288.246} C_VEL
LIN {X 0,Y 244.511,Z 215.342,A -85,B 0,C 180,E1 -20290.351,E2 -20290.351} C_VEL
LIN {X 0,Y 239.266,Z 206.056,A -85,B 0,C 180,E1 -20292.676,E2 -20292.676} C_VEL
LIN {X 0,Y 235.439,Z 200.065,A -85,B 0,C 180,E1 -20294.53,E2 -20294.53} C_VEL
LIN {X 0,Y 231.88,Z 194.651,A -85,B 0,C 180,E1 -20296.47,E2 -20296.47} C_VEL
LIN {X 0,Y 227.564,Z 188.531,A -85,B 0,C 180,E1 -20299.129,E2 -20299.129} C_VEL
LIN {X 0,Y 223.711,Z 183.42,A -85,B 0,C 180,E1 -20301.966,E2 -20301.966} C_VEL
LIN {X 0,Y 222.989,Z 182.015,A -85,B 0,C 180,E1 -20302.709,E2 -20302.709} C_VEL
LIN {X 0,Y 221.743,Z 178.594,A -85,B 0,C 180,E1 -20307.397,E2 -20307.397} C_VEL
LIN {X 0,Y 220.827,Z 175.966,A -85,B 0,C 180,E1 -20313.207,E2 -20313.207} C_VEL
LIN {X 0,Y 220.851,Z 175.963,A -85,B 0,C 180,E1 -20317.55,E2 -20317.55} C_VEL
LIN {X 0,Y 220.911,Z 175.964,A -85,B 0,C 180,E1 -20322.629,E2 -20322.629} C_VEL
LIN {X 0,Y 220.934,Z 176.018,A -85,B 0,C 180,E1 -20325.256,E2 -20325.256} C_VEL
LIN {X 0,Y 222.105,Z 178.645,A -85,B 0,C 180,E1 -20330.81,E2 -20330.81} C_VEL
LIN {X 0,Y 226.638,Z 184.104,A -85,B 0,C 180,E1 -20334.419,E2 -20334.419} C_VEL
LIN {X 0,Y 227.742,Z 185.566,A -85,B 0,C 180,E1 -20335.187,E2 -20335.187} C_VEL
LIN {X 0,Y 230.758,Z 189.04,A -85,B 0,C 180,E1 -20337.043,E2 -20337.043} C_VEL
LIN {X 0,Y 232.025,Z 190.509,A -85,B 0,C 180,E1 -20337.755,E2 -20337.755} C_VEL
LIN {X 0,Y 235.452,Z 195.3,A -85,B 0,C 180,E1 -20339.625,E2 -20339.625} C_VEL
LIN {X 0,Y 242.407,Z 206.13,A -85,B 0,C 180,E1 -20342.915,E2 -20342.915} C_VEL
LIN {X 0,Y 246.117,Z 212.476,A -85,B 0,C 180,E1 -20344.462,E2 -20344.462} C_VEL
LIN {X 0,Y 251.163,Z 222.363,A -85,B 0,C 180,E1 -20346.463,E2 -20346.463} C_VEL
LIN {X 0,Y 254.906,Z 230.965,A -85,B 0,C 180,E1 -20347.868,E2 -20347.868} C_VEL
LIN {X 0,Y 250.866,Z 285.349,A -85,B 0,C 180,E1 -20349.73,E2 -20349.73} C_VEL
LIN {X 0,Y 248.959,Z 299.331,A -85,B 0,C 180,E1 -20350.506,E2 -20350.506} C_VEL
LIN {X 0,Y 246.876,Z 311.183,A -85,B 0,C 180,E1 -20351.494,E2 -20351.494} C_VEL
LIN {X 0,Y 244.124,Z 323.313,A -85,B 0,C 180,E1 -20352.834,E2 -20352.834} C_VEL
LIN {X 0,Y 241.105,Z 334.042,A -85,B 0,C 180,E1 -20354.345,E2 -20354.345} C_VEL
LIN {X 0,Y 237.617,Z 344.86,A -85,B 0,C 180,E1 -20356.318,E2 -20356.318} C_VEL
LIN {X 0,Y 234.283,Z 353.76,A -85,B 0,C 180,E1 -20358.358,E2 -20358.358} C_VEL
LIN {X 0,Y 231.096,Z 361.772,A -85,B 0,C 180,E1 -20360.683,E2 -20360.683} C_VEL
LIN {X 0,Y 228.133,Z 368.498,A -85,B 0,C 180,E1 -20363.118,E2 -20363.118} C_VEL
LIN {X 0,Y 225.371,Z 374.426,A -85,B 0,C 180,E1 -20365.885,E2 -20365.885} C_VEL
LIN {X 0,Y 223.424,Z 378.403,A -85,B 0,C 180,E1 -20368.267,E2 -20368.267} C_VEL
LIN {X 0,Y 221.6,Z 381.94,A -85,B 0,C 180,E1 -20371.099,E2 -20371.099} C_VEL
LIN {X 0,Y 220.179,Z 384.362,A -85,B 0,C 180,E1 -20373.913,E2 -20373.913} C_VEL
LIN {X 0,Y 218.935,Z 386.004,A -85,B 0,C 180,E1 -20377.582,E2 -20377.582} C_VEL
LIN {X 0,Y 218.453,Z 386.239,A -85,B 0,C 180,E1 -20380.047,E2 -20380.047} C_VEL
LIN {X 0,Y 218.163,Z 385.72,A -85,B 0,C 180,E1 -20382.57,E2 -20382.57} C_VEL
LIN {X 0,Y 218.135,Z 384.394,A -85,B 0,C 180,E1 -20385.137,E2 -20385.137} C_VEL
LIN {X 0,Y 218.356,Z 382.218,A -85,B 0,C 180,E1 -20387.754,E2 -20387.754} C_VEL
LIN {X 0,Y 218.762,Z 379.044,A -85,B 0,C 180,E1 -20390.445,E2 -20390.445} C_VEL
LIN {X 0,Y 219.435,Z 374.711,A -85,B 0,C 180,E1 -20393.195,E2 -20393.195} C_VEL
LIN {X 0,Y 220.279,Z 368.903,A -85,B 0,C 180,E1 -20396.049,E2 -20396.049} C_VEL
LIN {X 0,Y 221.543,Z 361.458,A -85,B 0,C 180,E1 -20398.926,E2 -20398.926} C_VEL
LIN {X 0,Y 223.11,Z 352.727,A -85,B 0,C 180,E1 -20401.574,E2 -20401.574} C_VEL
LIN {X 0,Y 224.953,Z 342.427,A -85,B 0,C 180,E1 -20404.063,E2 -20404.063} C_VEL
LIN {X 0,Y 226.654,Z 332.39,A -85,B 0,C 180,E1 -20405.986,E2 -20405.986} C_VEL
LIN {X 0,Y 228.41,Z 320.396,A -85,B 0,C 180,E1 -20407.809,E2 -20407.809} C_VEL
LIN {X 0,Y 229.956,Z 308.623,A -85,B 0,C 180,E1 -20409.19,E2 -20409.19} C_VEL
LIN {X 0,Y 231.237,Z 295.661,A -85,B 0,C 180,E1 -20410.314,E2 -20410.314} C_VEL
LIN {X 0,Y 232.266,Z 281.926,A -85,B 0,C 180,E1 -20411.124,E2 -20411.124} C_VEL
LIN {X 0,Y 235.223,Z 215.237,A -85,B 0,C 180,E1 -20413.455,E2 -20413.455} C_VEL
LIN {X 0,Y 229.344,Z 197.664,A -85,B 0,C 180,E1 -20414.732,E2 -20414.732} C_VEL
LIN {X 0,Y 223.11,Z 181.343,A -85,B 0,C 180,E1 -20416.076,E2 -20416.076} C_VEL
LIN {X 0,Y 221.086,Z 176.546,A -85,B 0,C 180,E1 -20416.512,E2 -20416.512} C_VEL
LIN {X 0,Y 220.968,Z 175.964,A -85,B 0,C 180,E1 -20416.61,E2 -20416.61} C_VEL
LIN {X 0,Y 221.177,Z 175.932,A -85,B 0,C 180,E1 -20420.859,E2 -20420.859} C_VEL
LIN {X 0,Y 221.231,Z 175.928,A -85,B 0,C 180,E1 -20422.7,E2 -20422.7} C_VEL
LIN {X 0,Y 221.465,Z 175.902,A -85,B 0,C 180,E1 -20428.182,E2 -20428.182} C_VEL
LIN {X 0,Y 221.462,Z 175.902,A -85,B 0,C 180,E1 -20431.819,E2 -20431.819} C_VEL
LIN {X 0,Y 221.238,Z 175.927,A -85,B 0,C 180,E1 -20437.3,E2 -20437.3} C_VEL
LIN {X 0,Y 221.047,Z 175.951,A -85,B 0,C 180,E1 -20440.998,E2 -20440.998} C_VEL
LIN {X 0,Y 220.967,Z 175.958,A -85,B 0,C 180,E1 -20446.634,E2 -20446.634} C_VEL
LIN {X 0,Y 220.843,Z 175.973,A -85,B 0,C 180,E1 -20450.491,E2 -20450.491} C_VEL
LIN {X 0,Y 220.792,Z 175.979,A -85,B 0,C 180,E1 -20454.444,E2 -20454.444} C_VEL
LIN {X 0,Y 220.792,Z 175.98,A -85,B 0,C 180,E1 -20458.52,E2 -20458.52} C_VEL
LIN {X 0,Y 220.808,Z 175.971,A -85,B 0,C 180,E1 -20462.757,E2 -20462.757} C_VEL
LIN {X 0,Y 220.799,Z 175.983,A -85,B 0,C 180,E1 -20467.275,E2 -20467.275} C_VEL
LIN {X 0,Y 220.744,Z 175.978,A -85,B 0,C 180,E1 -20471.958,E2 -20471.958} C_VEL
LIN {X 0,Y 220.749,Z 175.982,A -85,B 0,C 180,E1 -20475.541,E2 -20475.541} C_VEL
LIN {X 0,Y 220.778,Z 175.983,A -85,B 0,C 180,E1 -20480.458,E2 -20480.458} C_VEL
LIN {X 0,Y 220.822,Z 175.976,A -85,B 0,C 180,E1 -20482.793,E2 -20482.793} C_VEL
LIN {X 0,Y 220.809,Z 175.967,A -85,B 0,C 180,E1 -20487.244,E2 -20487.244} C_VEL
LIN {X 0,Y 220.796,Z 175.978,A -85,B 0,C 180,E1 -20491.482,E2 -20491.482} C_VEL
LIN {X 0,Y 220.793,Z 175.979,A -85,B 0,C 180,E1 -20495.557,E2 -20495.557} C_VEL
LIN {X 0,Y 220.842,Z 175.965,A -85,B 0,C 180,E1 -20499.51,E2 -20499.51} C_VEL
LIN {X 0,Y 220.963,Z 175.949,A -85,B 0,C 180,E1 -20503.367,E2 -20503.367} C_VEL
LIN {X 0,Y 221.047,Z 175.947,A -85,B 0,C 180,E1 -20509.003,E2 -20509.003} C_VEL
LIN {X 0,Y 221.227,Z 175.918,A -85,B 0,C 180,E1 -20512.7,E2 -20512.7} C_VEL
LIN {X 0,Y 221.461,Z 175.894,A -85,B 0,C 180,E1 -20518.182,E2 -20518.182} C_VEL
LIN {X 0,Y 221.461,Z 175.898,A -85,B 0,C 180,E1 -20521.819,E2 -20521.819} C_VEL
LIN {X 0,Y 221.227,Z 175.916,A -85,B 0,C 180,E1 -20527.301,E2 -20527.301} C_VEL
LIN {X 0,Y 221.048,Z 175.948,A -85,B 0,C 180,E1 -20530.998,E2 -20530.998} C_VEL
LIN {X 0,Y 220.968,Z 175.951,A -85,B 0,C 180,E1 -20536.634,E2 -20536.634} C_VEL
LIN {X 0,Y 220.844,Z 175.975,A -85,B 0,C 180,E1 -20540.492,E2 -20540.492} C_VEL
LIN {X 0,Y 220.794,Z 175.976,A -85,B 0,C 180,E1 -20544.444,E2 -20544.444} C_VEL
LIN {X 0,Y 220.791,Z 175.983,A -85,B 0,C 180,E1 -20548.521,E2 -20548.521} C_VEL
LIN {X 0,Y 220.811,Z 175.97,A -85,B 0,C 180,E1 -20552.758,E2 -20552.758} C_VEL
LIN {X 0,Y 220.802,Z 175.982,A -85,B 0,C 180,E1 -20557.276,E2 -20557.276} C_VEL
LIN {X 0,Y 220.748,Z 175.987,A -85,B 0,C 180,E1 -20561.959,E2 -20561.959} C_VEL
LIN {X 0,Y 220.752,Z 175.987,A -85,B 0,C 180,E1 -20564.436,E2 -20564.436} C_VEL
LIN {X 0,Y 220.12,Z 176.072,A -85,B 0,C 180,E1 -20565.959,E2 -20565.959} C_VEL
LIN {X 0,Y 217.197,Z 176.435,A -85,B 0,C 180,E1 -20568.441,E2 -20568.441} C_VEL
LIN {X 0,Y 214.749,Z 176.736,A -85,B 0,C 180,E1 -20570.47,E2 -20570.47} C_VEL
LIN {X 0,Y 213.8,Z 176.853,A -85,B 0,C 180,E1 -20572.048,E2 -20572.048} C_VEL
LIN {X 0,Y 213.78,Z 176.857,A -85,B 0,C 180,E1 -20572.582,E2 -20572.582} C_VEL
LIN {X 0,Y 215.773,Z 186.128,A -85,B 0,C 180,E1 -20576.792,E2 -20576.792} C_VEL
LIN {X 0,Y 223.722,Z 208.646,A -85,B 0,C 180,E1 -20578.658,E2 -20578.658} C_VEL
LIN {X 0,Y 224.747,Z 212.602,A -85,B 0,C 180,E1 -20578.93,E2 -20578.93} C_VEL
LIN {X 0,Y 227.902,Z 237.698,A -85,B 0,C 180,E1 -20580.267,E2 -20580.267} C_VEL
LIN {X 0,Y 225.307,Z 294.897,A -85,B 0,C 180,E1 -20582.355,E2 -20582.355} C_VEL
LIN {X 0,Y 224.171,Z 308.738,A -85,B 0,C 180,E1 -20583.213,E2 -20583.213} C_VEL
LIN {X 0,Y 222.824,Z 320.813,A -85,B 0,C 180,E1 -20584.299,E2 -20584.299} C_VEL
LIN {X 0,Y 220.846,Z 333.332,A -85,B 0,C 180,E1 -20585.813,E2 -20585.813} C_VEL
LIN {X 0,Y 218.991,Z 344.639,A -85,B 0,C 180,E1 -20587.598,E2 -20587.598} C_VEL
LIN {X 0,Y 217.266,Z 354.471,A -85,B 0,C 180,E1 -20589.553,E2 -20589.553} C_VEL
LIN {X 0,Y 215.936,Z 362.454,A -85,B 0,C 180,E1 -20591.498,E2 -20591.498} C_VEL
LIN {X 0,Y 214.248,Z 371.742,A -85,B 0,C 180,E1 -20594.298,E2 -20594.298} C_VEL
LIN {X 0,Y 212.897,Z 379.193,A -85,B 0,C 180,E1 -20597.125,E2 -20597.125} C_VEL
LIN {X 0,Y 212.222,Z 384.225,A -85,B 0,C 180,E1 -20599.505,E2 -20599.505} C_VEL
LIN {X 0,Y 211.718,Z 389.074,A -85,B 0,C 180,E1 -20602.37,E2 -20602.37} C_VEL
LIN {X 0,Y 211.448,Z 393.213,A -85,B 0,C 180,E1 -20605.664,E2 -20605.664} C_VEL
LIN {X 0,Y 211.522,Z 395.337,A -85,B 0,C 180,E1 -20608.096,E2 -20608.096} C_VEL
LIN {X 0,Y 211.603,Z 396.533,A -85,B 0,C 180,E1 -20610,E2 -20610} C_VEL
LIN {X 0,Y 211.47,Z 397.26,A -85,B 0,C 180,E1 -20611.904,E2 -20611.904} C_VEL
LIN {X 0,Y 211.422,Z 397.599,A -85,B 0,C 180,E1 -20614.241,E2 -20614.241} C_VEL
LIN {X 0,Y 211.699,Z 397.044,A -85,B 0,C 180,E1 -20617.631,E2 -20617.631} C_VEL
LIN {X 0,Y 212.113,Z 396.172,A -85,B 0,C 180,E1 -20619.535,E2 -20619.535} C_VEL
LIN {X 0,Y 213.514,Z 393.195,A -85,B 0,C 180,E1 -20623.321,E2 -20623.321} C_VEL
LIN {X 0,Y 215.076,Z 389.85,A -85,B 0,C 180,E1 -20626.126,E2 -20626.126} C_VEL
LIN {X 0,Y 217.338,Z 385.449,A -85,B 0,C 180,E1 -20628.866,E2 -20628.866} C_VEL
LIN {X 0,Y 219.959,Z 379.928,A -85,B 0,C 180,E1 -20631.553,E2 -20631.553} C_VEL
LIN {X 0,Y 222.949,Z 373.088,A -85,B 0,C 180,E1 -20634.191,E2 -20634.191} C_VEL
LIN {X 0,Y 226.63,Z 364.624,A -85,B 0,C 180,E1 -20636.721,E2 -20636.721} C_VEL
LIN {X 0,Y 230.04,Z 355.994,A -85,B 0,C 180,E1 -20638.762,E2 -20638.762} C_VEL
LIN {X 0,Y 233.793,Z 345.463,A -85,B 0,C 180,E1 -20640.732,E2 -20640.732} C_VEL
LIN {X 0,Y 237.42,Z 333.696,A -85,B 0,C 180,E1 -20642.447,E2 -20642.447} C_VEL
LIN {X 0,Y 240.508,Z 322.055,A -85,B 0,C 180,E1 -20643.724,E2 -20643.724} C_VEL
LIN {X 0,Y 243.263,Z 309.058,A -85,B 0,C 180,E1 -20644.79,E2 -20644.79} C_VEL
LIN {X 0,Y 245.354,Z 295.405,A -85,B 0,C 180,E1 -20645.548,E2 -20645.548} C_VEL
LIN {X 0,Y 247.272,Z 272.253,A -85,B 0,C 180,E1 -20646.383,E2 -20646.383} C_VEL
LIN {X 0,Y 249.371,Z 243.84,A -85,B 0,C 180,E1 -20647.351,E2 -20647.351} C_VEL
LIN {X 0,Y 248.678,Z 238.261,A -85,B 0,C 180,E1 -20647.831,E2 -20647.831} C_VEL
LIN {X 0,Y 245.204,Z 229.601,A -85,B 0,C 180,E1 -20649.296,E2 -20649.296} C_VEL
LIN {X 0,Y 240.664,Z 219.957,A -85,B 0,C 180,E1 -20651.285,E2 -20651.285} C_VEL
LIN {X 0,Y 235.997,Z 211.408,A -85,B 0,C 180,E1 -20653.517,E2 -20653.517} C_VEL
LIN {X 0,Y 232.515,Z 205.733,A -85,B 0,C 180,E1 -20655.315,E2 -20655.315} C_VEL
LIN {X 0,Y 229.372,Z 200.755,A -85,B 0,C 180,E1 -20657.134,E2 -20657.134} C_VEL
LIN {X 0,Y 225.356,Z 194.831,A -85,B 0,C 180,E1 -20659.76,E2 -20659.76} C_VEL
LIN {X 0,Y 221.788,Z 189.892,A -85,B 0,C 180,E1 -20662.531,E2 -20662.531} C_VEL
LIN {X 0,Y 220.892,Z 188.42,A -85,B 0,C 180,E1 -20663.375,E2 -20663.375} C_VEL
LIN {X 0,Y 215.957,Z 182.429,A -85,B 0,C 180,E1 -20669.126,E2 -20669.126} C_VEL
LIN {X 0,Y 215.189,Z 181.053,A -85,B 0,C 180,E1 -20670.665,E2 -20670.665} C_VEL
LIN {X 0,Y 215.035,Z 180.188,A -85,B 0,C 180,E1 -20672.769,E2 -20672.769} C_VEL
LIN {X 0,Y 214.618,Z 179.388,A -85,B 0,C 180,E1 -20676.86,E2 -20676.86} C_VEL
LIN {X 0,Y 214.818,Z 179.579,A -85,B 0,C 180,E1 -20682.789,E2 -20682.789} C_VEL
LIN {X 0,Y 216.991,Z 182.405,A -85,B 0,C 180,E1 -20686.642,E2 -20686.642} C_VEL
LIN {X 0,Y 220.656,Z 185.67,A -85,B 0,C 180,E1 -20690.589,E2 -20690.589} C_VEL
LIN {X 0,Y 224.535,Z 190.532,A -85,B 0,C 180,E1 -20693.823,E2 -20693.823} C_VEL
LIN {X 0,Y 225.672,Z 192.007,A -85,B 0,C 180,E1 -20694.638,E2 -20694.638} C_VEL
LIN {X 0,Y 228.739,Z 195.648,A -85,B 0,C 180,E1 -20696.627,E2 -20696.627} C_VEL
LIN {X 0,Y 232.766,Z 201.225,A -85,B 0,C 180,E1 -20698.937,E2 -20698.937} C_VEL
LIN {X 0,Y 239.559,Z 212.221,A -85,B 0,C 180,E1 -20702.333,E2 -20702.333} C_VEL
LIN {X 0,Y 244.167,Z 220.645,A -85,B 0,C 180,E1 -20704.354,E2 -20704.354} C_VEL
LIN {X 0,Y 248.983,Z 231.062,A -85,B 0,C 180,E1 -20706.355,E2 -20706.355} C_VEL
LIN {X 0,Y 250.033,Z 233.623,A -85,B 0,C 180,E1 -20706.77,E2 -20706.77} C_VEL
LIN {X 0,Y 245.929,Z 285.542,A -85,B 0,C 180,E1 -20708.55,E2 -20708.55} C_VEL
LIN {X 0,Y 243.989,Z 299.32,A -85,B 0,C 180,E1 -20709.324,E2 -20709.324} C_VEL
LIN {X 0,Y 241.677,Z 311.671,A -85,B 0,C 180,E1 -20710.365,E2 -20710.365} C_VEL
LIN {X 0,Y 238.885,Z 323.293,A -85,B 0,C 180,E1 -20711.669,E2 -20711.669} C_VEL
LIN {X 0,Y 235.683,Z 334.186,A -85,B 0,C 180,E1 -20713.229,E2 -20713.229} C_VEL
LIN {X 0,Y 232.455,Z 343.803,A -85,B 0,C 180,E1 -20714.969,E2 -20714.969} C_VEL
LIN {X 0,Y 228.912,Z 352.903,A -85,B 0,C 180,E1 -20717.028,E2 -20717.028} C_VEL
LIN {X 0,Y 225.218,Z 361.684,A -85,B 0,C 180,E1 -20719.572,E2 -20719.572} C_VEL
LIN {X 0,Y 221.704,Z 369.165,A -85,B 0,C 180,E1 -20722.358,E2 -20722.358} C_VEL
LIN {X 0,Y 219.316,Z 373.924,A -85,B 0,C 180,E1 -20724.618,E2 -20724.618} C_VEL
LIN {X 0,Y 216.64,Z 378.99,A -85,B 0,C 180,E1 -20727.738,E2 -20727.738} C_VEL
LIN {X 0,Y 214.878,Z 382.152,A -85,B 0,C 180,E1 -20730.369,E2 -20730.369} C_VEL
LIN {X 0,Y 212.973,Z 385.068,A -85,B 0,C 180,E1 -20734.123,E2 -20734.123} C_VEL
LIN {X 0,Y 211.906,Z 386.259,A -85,B 0,C 180,E1 -20737.254,E2 -20737.254} C_VEL
LIN {X 0,Y 211.349,Z 386.39,A -85,B 0,C 180,E1 -20740.111,E2 -20740.111} C_VEL
LIN {X 0,Y 211.051,Z 385.66,A -85,B 0,C 180,E1 -20742.897,E2 -20742.897} C_VEL
LIN {X 0,Y 211.053,Z 384.106,A -85,B 0,C 180,E1 -20745.631,E2 -20745.631} C_VEL
LIN {X 0,Y 211.34,Z 381.718,A -85,B 0,C 180,E1 -20748.312,E2 -20748.312} C_VEL
LIN {X 0,Y 211.74,Z 378.531,A -85,B 0,C 180,E1 -20750.904,E2 -20750.904} C_VEL
LIN {X 0,Y 212.543,Z 373.497,A -85,B 0,C 180,E1 -20754.018,E2 -20754.018} C_VEL
LIN {X 0,Y 213.563,Z 366.908,A -85,B 0,C 180,E1 -20757.114,E2 -20757.114} C_VEL
LIN {X 0,Y 215.057,Z 358.756,A -85,B 0,C 180,E1 -20760.109,E2 -20760.109} C_VEL
LIN {X 0,Y 216.754,Z 349.612,A -85,B 0,C 180,E1 -20762.756,E2 -20762.756} C_VEL
LIN {X 0,Y 218.407,Z 340.404,A -85,B 0,C 180,E1 -20764.899,E2 -20764.899} C_VEL
LIN {X 0,Y 220.369,Z 329.126,A -85,B 0,C 180,E1 -20767,E2 -20767} C_VEL
LIN {X 0,Y 221.966,Z 317.873,A -85,B 0,C 180,E1 -20768.647,E2 -20768.647} C_VEL
LIN {X 0,Y 223.673,Z 304.82,A -85,B 0,C 180,E1 -20770.097,E2 -20770.097} C_VEL
LIN {X 0,Y 224.819,Z 291.935,A -85,B 0,C 180,E1 -20771.141,E2 -20771.141} C_VEL
LIN {X 0,Y 225.805,Z 278.528,A -85,B 0,C 180,E1 -20771.837,E2 -20771.837} C_VEL
LIN {X 0,Y 228.579,Z 216.657,A -85,B 0,C 180,E1 -20774.051,E2 -20774.051} C_VEL
LIN {X 0,Y 221.744,Z 196.388,A -85,B 0,C 180,E1 -20775.603,E2 -20775.603} C_VEL
LIN {X 0,Y 216.593,Z 183.287,A -85,B 0,C 180,E1 -20776.761,E2 -20776.761} C_VEL
LIN {X 0,Y 214.081,Z 177.546,A -85,B 0,C 180,E1 -20777.318,E2 -20777.318} C_VEL
LIN {X 0,Y 213.936,Z 176.84,A -85,B 0,C 180,E1 -20777.43,E2 -20777.43} C_VEL
LIN {X 0,Y 214.118,Z 176.812,A -85,B 0,C 180,E1 -20780.555,E2 -20780.555} C_VEL
LIN {X 0,Y 214.07,Z 176.821,A -85,B 0,C 180,E1 -20784.348,E2 -20784.348} C_VEL
LIN {X 0,Y 214.401,Z 176.782,A -85,B 0,C 180,E1 -20788.122,E2 -20788.122} C_VEL
LIN {X 0,Y 214.509,Z 176.769,A -85,B 0,C 180,E1 -20790,E2 -20790} C_VEL
LIN {X 0,Y 214.399,Z 176.782,A -85,B 0,C 180,E1 -20791.879,E2 -20791.879} C_VEL
LIN {X 0,Y 214.18,Z 176.808,A -85,B 0,C 180,E1 -20797.542,E2 -20797.542} C_VEL
LIN {X 0,Y 213.979,Z 176.833,A -85,B 0,C 180,E1 -20801.366,E2 -20801.366} C_VEL
LIN {X 0,Y 213.868,Z 176.846,A -85,B 0,C 180,E1 -20805.242,E2 -20805.242} C_VEL
LIN {X 0,Y 213.787,Z 176.855,A -85,B 0,C 180,E1 -20809.192,E2 -20809.192} C_VEL
LIN {X 0,Y 213.761,Z 176.858,A -85,B 0,C 180,E1 -20813.237,E2 -20813.237} C_VEL
LIN {X 0,Y 213.782,Z 176.857,A -85,B 0,C 180,E1 -20817.427,E2 -20817.427} C_VEL
LIN {X 0,Y 213.755,Z 176.849,A -85,B 0,C 180,E1 -20821.739,E2 -20821.739} C_VEL
LIN {X 0,Y 213.738,Z 176.859,A -85,B 0,C 180,E1 -20826.289,E2 -20826.289} C_VEL
LIN {X 0,Y 213.694,Z 176.859,A -85,B 0,C 180,E1 -20831.129,E2 -20831.129} C_VEL
LIN {X 0,Y 213.698,Z 176.854,A -85,B 0,C 180,E1 -20833.68,E2 -20833.68} C_VEL
LIN {X 0,Y 213.698,Z 176.86,A -85,B 0,C 180,E1 -20836.346,E2 -20836.346} C_VEL
LIN {X 0,Y 213.701,Z 176.863,A -85,B 0,C 180,E1 -20841.33,E2 -20841.33} C_VEL
LIN {X 0,Y 213.751,Z 176.844,A -85,B 0,C 180,E1 -20846.018,E2 -20846.018} C_VEL
LIN {X 0,Y 213.745,Z 176.854,A -85,B 0,C 180,E1 -20850.45,E2 -20850.45} C_VEL
LIN {X 0,Y 213.744,Z 176.861,A -85,B 0,C 180,E1 -20854.695,E2 -20854.695} C_VEL
LIN {X 0,Y 213.771,Z 176.847,A -85,B 0,C 180,E1 -20858.8,E2 -20858.8} C_VEL
LIN {X 0,Y 213.875,Z 176.831,A -85,B 0,C 180,E1 -20862.799,E2 -20862.799} C_VEL
LIN {X 0,Y 213.907,Z 176.837,A -85,B 0,C 180,E1 -20866.704,E2 -20866.704} C_VEL
LIN {X 0,Y 214.12,Z 176.809,A -85,B 0,C 180,E1 -20870.555,E2 -20870.555} C_VEL
LIN {X 0,Y 214.063,Z 176.805,A -85,B 0,C 180,E1 -20874.348,E2 -20874.348} C_VEL
LIN {X 0,Y 214.398,Z 176.773,A -85,B 0,C 180,E1 -20878.122,E2 -20878.122} C_VEL
LIN {X 0,Y 214.509,Z 176.763,A -85,B 0,C 180,E1 -20880.001,E2 -20880.001} C_VEL
LIN {X 0,Y 214.398,Z 176.778,A -85,B 0,C 180,E1 -20881.879,E2 -20881.879} C_VEL
LIN {X 0,Y 214.169,Z 176.795,A -85,B 0,C 180,E1 -20887.543,E2 -20887.543} C_VEL
LIN {X 0,Y 213.98,Z 176.829,A -85,B 0,C 180,E1 -20891.366,E2 -20891.366} C_VEL
LIN {X 0,Y 213.869,Z 176.841,A -85,B 0,C 180,E1 -20895.242,E2 -20895.242} C_VEL
LIN {X 0,Y 213.788,Z 176.853,A -85,B 0,C 180,E1 -20899.193,E2 -20899.193} C_VEL
LIN {X 0,Y 213.763,Z 176.857,A -85,B 0,C 180,E1 -20903.237,E2 -20903.237} C_VEL
LIN {X 0,Y 213.766,Z 176.86,A -85,B 0,C 180,E1 -20907.418,E2 -20907.418} C_VEL
LIN {X 0,Y 213.758,Z 176.85,A -85,B 0,C 180,E1 -20911.74,E2 -20911.74} C_VEL
LIN {X 0,Y 213.742,Z 176.857,A -85,B 0,C 180,E1 -20916.29,E2 -20916.29} C_VEL
LIN {X 0,Y 213.698,Z 176.867,A -85,B 0,C 180,E1 -20921.129,E2 -20921.129} C_VEL
LIN {X 0,Y 213.656,Z 176.866,A -85,B 0,C 180,E1 -20924.418,E2 -20924.418} C_VEL
LIN {X 0,Y 213.699,Z 176.867,A -85,B 0,C 180,E1 -20928.872,E2 -20928.872} C_VEL
LIN {X 0,Y 213.78,Z 176.857,A -85,B 0,C 180,E1 -20932.582,E2 -20932.582} C_VEL
LIN {X 0,Y 213.395,Z 179.369,A -85,B 0,C 180,E1 -20933.627,E2 -20933.627} C_VEL
LIN {X 0,Y 211.383,Z 183.61,A -85,B 0,C 180,E1 -20935.13,E2 -20935.13} C_VEL
LIN {X 0,Y 210.342,Z 188.632,A -85,B 0,C 180,E1 -20936.043,E2 -20936.043} C_VEL
LIN {X 0,Y 210.866,Z 192.247,A -85,B 0,C 180,E1 -20936.478,E2 -20936.478} C_VEL
LIN {X 0,Y 218.156,Z 213.206,A -85,B 0,C 180,E1 -20938.242,E2 -20938.242} C_VEL
LIN {X 0,Y 221.242,Z 238.274,A -85,B 0,C 180,E1 -20939.627,E2 -20939.627} C_VEL
LIN {X 0,Y 218.683,Z 293.742,A -85,B 0,C 180,E1 -20941.704,E2 -20941.704} C_VEL
LIN {X 0,Y 217.588,Z 307.16,A -85,B 0,C 180,E1 -20942.53,E2 -20942.53} C_VEL
LIN {X 0,Y 216.112,Z 320.121,A -85,B 0,C 180,E1 -20943.699,E2 -20943.699} C_VEL
LIN {X 0,Y 214.39,Z 331.213,A -85,B 0,C 180,E1 -20945.035,E2 -20945.035} C_VEL
LIN {X 0,Y 212.456,Z 342.864,A -85,B 0,C 180,E1 -20946.87,E2 -20946.87} C_VEL
LIN {X 0,Y 210.458,Z 353.586,A -85,B 0,C 180,E1 -20949.007,E2 -20949.007} C_VEL
LIN {X 0,Y 209.085,Z 361.141,A -85,B 0,C 180,E1 -20950.869,E2 -20950.869} C_VEL
LIN {X 0,Y 207.638,Z 369.27,A -85,B 0,C 180,E1 -20953.279,E2 -20953.279} C_VEL
LIN {X 0,Y 206.13,Z 377.159,A -85,B 0,C 180,E1 -20956.192,E2 -20956.192} C_VEL
LIN {X 0,Y 205.198,Z 383.467,A -85,B 0,C 180,E1 -20959.142,E2 -20959.142} C_VEL
LIN {X 0,Y 204.661,Z 388.438,A -85,B 0,C 180,E1 -20962.105,E2 -20962.105} C_VEL
LIN {X 0,Y 204.494,Z 391.103,A -85,B 0,C 180,E1 -20964.082,E2 -20964.082} C_VEL
LIN {X 0,Y 204.367,Z 393.241,A -85,B 0,C 180,E1 -20966.056,E2 -20966.056} C_VEL
LIN {X 0,Y 204.421,Z 394.911,A -85,B 0,C 180,E1 -20968.029,E2 -20968.029} C_VEL
LIN {X 0,Y 204.517,Z 396.157,A -85,B 0,C 180,E1 -20970,E2 -20970} C_VEL
LIN {X 0,Y 204.372,Z 396.974,A -85,B 0,C 180,E1 -20971.97,E2 -20971.97} C_VEL
LIN {X 0,Y 204.324,Z 397.355,A -85,B 0,C 180,E1 -20974.045,E2 -20974.045} C_VEL
LIN {X 0,Y 204.652,Z 396.924,A -85,B 0,C 180,E1 -20977.895,E2 -20977.895} C_VEL
LIN {X 0,Y 205.103,Z 396.136,A -85,B 0,C 180,E1 -20979.865,E2 -20979.865} C_VEL
LIN {X 0,Y 205.739,Z 394.921,A -85,B 0,C 180,E1 -20981.827,E2 -20981.827} C_VEL
LIN {X 0,Y 207.586,Z 391.256,A -85,B 0,C 180,E1 -20985.714,E2 -20985.714} C_VEL
LIN {X 0,Y 209.789,Z 387.359,A -85,B 0,C 180,E1 -20988.557,E2 -20988.557} C_VEL
LIN {X 0,Y 212.533,Z 382.363,A -85,B 0,C 180,E1 -20991.33,E2 -20991.33} C_VEL
LIN {X 0,Y 214.867,Z 377.172,A -85,B 0,C 180,E1 -20993.673,E2 -20993.673} C_VEL
LIN {X 0,Y 218.408,Z 369.849,A -85,B 0,C 180,E1 -20996.26,E2 -20996.26} C_VEL
LIN {X 0,Y 221.709,Z 362.346,A -85,B 0,C 180,E1 -20998.39,E2 -20998.39} C_VEL
LIN {X 0,Y 225.905,Z 352.357,A -85,B 0,C 180,E1 -21000.625,E2 -21000.625} C_VEL
LIN {X 0,Y 229.884,Z 341.052,A -85,B 0,C 180,E1 -21002.603,E2 -21002.603} C_VEL
LIN {X 0,Y 233.349,Z 329.788,A -85,B 0,C 180,E1 -21004.12,E2 -21004.12} C_VEL
LIN {X 0,Y 236.62,Z 317.028,A -85,B 0,C 180,E1 -21005.392,E2 -21005.392} C_VEL
LIN {X 0,Y 239.278,Z 303.697,A -85,B 0,C 180,E1 -21006.349,E2 -21006.349} C_VEL
LIN {X 0,Y 241.102,Z 290.156,A -85,B 0,C 180,E1 -21006.992,E2 -21006.992} C_VEL
LIN {X 0,Y 244.625,Z 244.965,A -85,B 0,C 180,E1 -21008.577,E2 -21008.577} C_VEL
LIN {X 0,Y 244.174,Z 241.317,A -85,B 0,C 180,E1 -21008.918,E2 -21008.918} C_VEL
LIN {X 0,Y 240.33,Z 231.908,A -85,B 0,C 180,E1 -21010.649,E2 -21010.649} C_VEL
LIN {X 0,Y 236.516,Z 223.743,A -85,B 0,C 180,E1 -21012.471,E2 -21012.471} C_VEL
LIN {X 0,Y 232.468,Z 216.261,A -85,B 0,C 180,E1 -21014.535,E2 -21014.535} C_VEL
LIN {X 0,Y 229.624,Z 211.323,A -85,B 0,C 180,E1 -21016.153,E2 -21016.153} C_VEL
LIN {X 0,Y 226.906,Z 206.847,A -85,B 0,C 180,E1 -21017.809,E2 -21017.809} C_VEL
LIN {X 0,Y 223.11,Z 201.049,A -85,B 0,C 180,E1 -21020.458,E2 -21020.458} C_VEL
LIN {X 0,Y 219.678,Z 195.917,A -85,B 0,C 180,E1 -21023.354,E2 -21023.354} C_VEL
LIN {X 0,Y 218.744,Z 194.707,A -85,B 0,C 180,E1 -21024.242,E2 -21024.242} C_VEL
LIN {X 0,Y 214.519,Z 189.106,A -85,B 0,C 180,E1 -21029.637,E2 -21029.637} C_VEL
LIN {X 0,Y 213.547,Z 187.572,A -85,B 0,C 180,E1 -21031.712,E2 -21031.712} C_VEL
LIN {X 0,Y 212.514,Z 186.322,A -85,B 0,C 180,E1 -21035.582,E2 -21035.582} C_VEL
LIN {X 0,Y 212.915,Z 186.246,A -85,B 0,C 180,E1 -21040.725,E2 -21040.725} C_VEL
LIN {X 0,Y 213.801,Z 186.786,A -85,B 0,C 180,E1 -21043.037,E2 -21043.037} C_VEL
LIN {X 0,Y 218.821,Z 192.117,A -85,B 0,C 180,E1 -21049.972,E2 -21049.972} C_VEL
LIN {X 0,Y 222.802,Z 197.271,A -85,B 0,C 180,E1 -21053.462,E2 -21053.462} C_VEL
LIN {X 0,Y 226.318,Z 201.848,A -85,B 0,C 180,E1 -21055.937,E2 -21055.937} C_VEL
LIN {X 0,Y 227.559,Z 203.525,A -85,B 0,C 180,E1 -21056.724,E2 -21056.724} C_VEL
LIN {X 0,Y 230.28,Z 207.542,A -85,B 0,C 180,E1 -21058.336,E2 -21058.336} C_VEL
LIN {X 0,Y 236.426,Z 217.76,A -85,B 0,C 180,E1 -21061.581,E2 -21061.581} C_VEL
LIN {X 0,Y 240.616,Z 225.844,A -85,B 0,C 180,E1 -21063.565,E2 -21063.565} C_VEL
LIN {X 0,Y 245.107,Z 235.888,A -85,B 0,C 180,E1 -21065.533,E2 -21065.533} C_VEL
LIN {X 0,Y 245.189,Z 237.583,A -85,B 0,C 180,E1 -21065.655,E2 -21065.655} C_VEL
LIN {X 0,Y 241.067,Z 286.102,A -85,B 0,C 180,E1 -21067.343,E2 -21067.343} C_VEL
LIN {X 0,Y 239.263,Z 298.645,A -85,B 0,C 180,E1 -21068.052,E2 -21068.052} C_VEL
LIN {X 0,Y 236.896,Z 310.978,A -85,B 0,C 180,E1 -21069.065,E2 -21069.065} C_VEL
LIN {X 0,Y 233.924,Z 322.876,A -85,B 0,C 180,E1 -21070.384,E2 -21070.384} C_VEL
LIN {X 0,Y 230.5,Z 334.084,A -85,B 0,C 180,E1 -21071.989,E2 -21071.989} C_VEL
LIN {X 0,Y 226.828,Z 344.415,A -85,B 0,C 180,E1 -21073.893,E2 -21073.893} C_VEL
LIN {X 0,Y 223.014,Z 353.605,A -85,B 0,C 180,E1 -21076.037,E2 -21076.037} C_VEL
LIN {X 0,Y 219.012,Z 362.542,A -85,B 0,C 180,E1 -21078.716,E2 -21078.716} C_VEL
LIN {X 0,Y 215.43,Z 369.646,A -85,B 0,C 180,E1 -21081.465,E2 -21081.465} C_VEL
LIN {X 0,Y 212.228,Z 375.534,A -85,B 0,C 180,E1 -21084.452,E2 -21084.452} C_VEL
LIN {X 0,Y 209.209,Z 380.722,A -85,B 0,C 180,E1 -21088.053,E2 -21088.053} C_VEL
LIN {X 0,Y 206.886,Z 384.278,A -85,B 0,C 180,E1 -21091.871,E2 -21091.871} C_VEL
LIN {X 0,Y 205.298,Z 386.207,A -85,B 0,C 180,E1 -21095.588,E2 -21095.588} C_VEL
LIN {X 0,Y 204.583,Z 386.647,A -85,B 0,C 180,E1 -21098.195,E2 -21098.195} C_VEL
LIN {X 0,Y 204.136,Z 386.404,A -85,B 0,C 180,E1 -21100.853,E2 -21100.853} C_VEL
LIN {X 0,Y 203.93,Z 385.374,A -85,B 0,C 180,E1 -21103.639,E2 -21103.639} C_VEL
LIN {X 0,Y 204.029,Z 383.468,A -85,B 0,C 180,E1 -21106.456,E2 -21106.456} C_VEL
LIN {X 0,Y 204.359,Z 380.761,A -85,B 0,C 180,E1 -21109.201,E2 -21109.201} C_VEL
LIN {X 0,Y 204.906,Z 376.949,A -85,B 0,C 180,E1 -21112.078,E2 -21112.078} C_VEL
LIN {X 0,Y 205.71,Z 371.777,A -85,B 0,C 180,E1 -21115.078,E2 -21115.078} C_VEL
LIN {X 0,Y 206.856,Z 365.025,A -85,B 0,C 180,E1 -21118.143,E2 -21118.143} C_VEL
LIN {X 0,Y 208.303,Z 357.4,A -85,B 0,C 180,E1 -21120.872,E2 -21120.872} C_VEL
LIN {X 0,Y 210.213,Z 347.454,A -85,B 0,C 180,E1 -21123.707,E2 -21123.707} C_VEL
LIN {X 0,Y 212.109,Z 337.011,A -85,B 0,C 180,E1 -21126.054,E2 -21126.054} C_VEL
LIN {X 0,Y 214.046,Z 325.628,A -85,B 0,C 180,E1 -21128.07,E2 -21128.07} C_VEL
LIN {X 0,Y 215.71,Z 314.111,A -85,B 0,C 180,E1 -21129.673,E2 -21129.673} C_VEL
LIN {X 0,Y 217.339,Z 300.755,A -85,B 0,C 180,E1 -21131.052,E2 -21131.052} C_VEL
LIN {X 0,Y 218.481,Z 287.508,A -85,B 0,C 180,E1 -21132.026,E2 -21132.026} C_VEL
LIN {X 0,Y 219.358,Z 272.211,A -85,B 0,C 180,E1 -21132.702,E2 -21132.702} C_VEL
LIN {X 0,Y 221.907,Z 217.504,A -85,B 0,C 180,E1 -21134.708,E2 -21134.708} C_VEL
LIN {X 0,Y 213.339,Z 192.964,A -85,B 0,C 180,E1 -21136.729,E2 -21136.729} C_VEL
LIN {X 0,Y 207.085,Z 178.567,A -85,B 0,C 180,E1 -21138.14,E2 -21138.14} C_VEL
LIN {X 0,Y 206.913,Z 177.713,A -85,B 0,C 180,E1 -21138.241,E2 -21138.241} C_VEL
LIN {X 0,Y 207.116,Z 177.685,A -85,B 0,C 180,E1 -21142.2,E2 -21142.2} C_VEL
LIN {X 0,Y 207.341,Z 177.661,A -85,B 0,C 180,E1 -21148.058,E2 -21148.058} C_VEL
LIN {X 0,Y 207.477,Z 177.645,A -85,B 0,C 180,E1 -21150,E2 -21150} C_VEL
LIN {X 0,Y 207.338,Z 177.662,A -85,B 0,C 180,E1 -21151.943,E2 -21151.943} C_VEL
LIN {X 0,Y 207.124,Z 177.688,A -85,B 0,C 180,E1 -21157.801,E2 -21157.801} C_VEL
LIN {X 0,Y 206.9,Z 177.717,A -85,B 0,C 180,E1 -21161.76,E2 -21161.76} C_VEL
LIN {X 0,Y 206.801,Z 177.726,A -85,B 0,C 180,E1 -21165.776,E2 -21165.776} C_VEL
LIN {X 0,Y 206.708,Z 177.736,A -85,B 0,C 180,E1 -21169.877,E2 -21169.877} C_VEL
LIN {X 0,Y 206.688,Z 177.737,A -85,B 0,C 180,E1 -21174.081,E2 -21174.081} C_VEL
LIN {X 0,Y 206.683,Z 177.737,A -85,B 0,C 180,E1 -21178.428,E2 -21178.428} C_VEL
LIN {X 0,Y 206.691,Z 177.729,A -85,B 0,C 180,E1 -21182.959,E2 -21182.959} C_VEL
LIN {X 0,Y 206.665,Z 177.741,A -85,B 0,C 180,E1 -21187.743,E2 -21187.743} C_VEL
LIN {X 0,Y 206.627,Z 177.736,A -85,B 0,C 180,E1 -21191.559,E2 -21191.559} C_VEL
LIN {X 0,Y 206.626,Z 177.741,A -85,B 0,C 180,E1 -21195.583,E2 -21195.583} C_VEL
LIN {X 0,Y 206.644,Z 177.743,A -85,B 0,C 180,E1 -21199.746,E2 -21199.746} C_VEL
LIN {X 0,Y 206.697,Z 177.727,A -85,B 0,C 180,E1 -21204.689,E2 -21204.689} C_VEL
LIN {X 0,Y 206.692,Z 177.731,A -85,B 0,C 180,E1 -21209.335,E2 -21209.335} C_VEL
LIN {X 0,Y 206.68,Z 177.738,A -85,B 0,C 180,E1 -21213.766,E2 -21213.766} C_VEL
LIN {X 0,Y 206.704,Z 177.732,A -85,B 0,C 180,E1 -21218.038,E2 -21218.038} C_VEL
LIN {X 0,Y 206.8,Z 177.706,A -85,B 0,C 180,E1 -21222.191,E2 -21222.191} C_VEL
LIN {X 0,Y 206.848,Z 177.715,A -85,B 0,C 180,E1 -21226.242,E2 -21226.242} C_VEL
LIN {X 0,Y 207.07,Z 177.689,A -85,B 0,C 180,E1 -21230.23,E2 -21230.23} C_VEL
LIN {X 0,Y 207.027,Z 177.682,A -85,B 0,C 180,E1 -21234.156,E2 -21234.156} C_VEL
LIN {X 0,Y 207.337,Z 177.651,A -85,B 0,C 180,E1 -21238.058,E2 -21238.058} C_VEL
LIN {X 0,Y 207.477,Z 177.639,A -85,B 0,C 180,E1 -21240.001,E2 -21240.001} C_VEL
LIN {X 0,Y 207.338,Z 177.658,A -85,B 0,C 180,E1 -21241.943,E2 -21241.943} C_VEL
LIN {X 0,Y 207.114,Z 177.675,A -85,B 0,C 180,E1 -21247.802,E2 -21247.802} C_VEL
LIN {X 0,Y 206.901,Z 177.714,A -85,B 0,C 180,E1 -21251.761,E2 -21251.761} C_VEL
LIN {X 0,Y 206.802,Z 177.718,A -85,B 0,C 180,E1 -21255.777,E2 -21255.777} C_VEL
LIN {X 0,Y 206.709,Z 177.738,A -85,B 0,C 180,E1 -21259.877,E2 -21259.877} C_VEL
LIN {X 0,Y 206.687,Z 177.734,A -85,B 0,C 180,E1 -21264.082,E2 -21264.082} C_VEL
LIN {X 0,Y 206.678,Z 177.741,A -85,B 0,C 180,E1 -21268.43,E2 -21268.43} C_VEL
LIN {X 0,Y 206.694,Z 177.725,A -85,B 0,C 180,E1 -21272.959,E2 -21272.959} C_VEL
LIN {X 0,Y 206.668,Z 177.741,A -85,B 0,C 180,E1 -21277.743,E2 -21277.743} C_VEL
LIN {X 0,Y 206.631,Z 177.747,A -85,B 0,C 180,E1 -21281.56,E2 -21281.56} C_VEL
LIN {X 0,Y 206.63,Z 177.746,A -85,B 0,C 180,E1 -21285.584,E2 -21285.584} C_VEL
LIN {X 0,Y 206.649,Z 177.744,A -85,B 0,C 180,E1 -21289.746,E2 -21289.746} C_VEL
LIN {X 0,Y 206.691,Z 177.816,A -85,B 0,C 180,E1 -21292.062,E2 -21292.062} C_VEL
LIN {X 0,Y 208.489,Z 185.968,A -85,B 0,C 180,E1 -21295.902,E2 -21295.902} C_VEL
LIN {X 0,Y 210.866,Z 192.247,A -85,B 0,C 180,E1 -21296.478,E2 -21296.478} C_VEL
LIN {X 0,Y 212.2,Z 197.816,A -85,B 0,C 180,E1 -21296.885,E2 -21296.885} C_VEL
LIN {X 0,Y 212.631,Z 207.576,A -85,B 0,C 180,E1 -21297.364,E2 -21297.364} C_VEL
LIN {X 0,Y 212.433,Z 215.553,A -85,B 0,C 180,E1 -21297.692,E2 -21297.692} C_VEL
LIN {X 0,Y 212.833,Z 223.454,A -85,B 0,C 180,E1 -21298.082,E2 -21298.082} C_VEL
LIN {X 0,Y 214.627,Z 239.979,A -85,B 0,C 180,E1 -21298.999,E2 -21298.999} C_VEL
LIN {X 0,Y 211.925,Z 294.722,A -85,B 0,C 180,E1 -21301.123,E2 -21301.123} C_VEL
LIN {X 0,Y 210.724,Z 308.476,A -85,B 0,C 180,E1 -21302.03,E2 -21302.03} C_VEL
LIN {X 0,Y 209.114,Z 321.478,A -85,B 0,C 180,E1 -21303.288,E2 -21303.288} C_VEL
LIN {X 0,Y 207.065,Z 333.761,A -85,B 0,C 180,E1 -21304.896,E2 -21304.896} C_VEL
LIN {X 0,Y 205.081,Z 344.899,A -85,B 0,C 180,E1 -21306.79,E2 -21306.79} C_VEL
LIN {X 0,Y 203.344,Z 354.385,A -85,B 0,C 180,E1 -21308.827,E2 -21308.827} C_VEL
LIN {X 0,Y 201.735,Z 363.326,A -85,B 0,C 180,E1 -21311.201,E2 -21311.201} C_VEL
LIN {X 0,Y 199.992,Z 372.389,A -85,B 0,C 180,E1 -21314.196,E2 -21314.196} C_VEL
LIN {X 0,Y 198.651,Z 379.625,A -85,B 0,C 180,E1 -21317.225,E2 -21317.225} C_VEL
LIN {X 0,Y 197.789,Z 386.196,A -85,B 0,C 180,E1 -21320.799,E2 -21320.799} C_VEL
LIN {X 0,Y 197.433,Z 390.482,A -85,B 0,C 180,E1 -21323.869,E2 -21323.869} C_VEL
LIN {X 0,Y 197.288,Z 392.725,A -85,B 0,C 180,E1 -21325.914,E2 -21325.914} C_VEL
LIN {X 0,Y 197.323,Z 394.465,A -85,B 0,C 180,E1 -21327.959,E2 -21327.959} C_VEL
LIN {X 0,Y 197.434,Z 395.768,A -85,B 0,C 180,E1 -21330,E2 -21330} C_VEL
LIN {X 0,Y 197.25,Z 397.095,A -85,B 0,C 180,E1 -21333.93,E2 -21333.93} C_VEL
LIN {X 0,Y 197.345,Z 397.156,A -85,B 0,C 180,E1 -21336.133,E2 -21336.133} C_VEL
LIN {X 0,Y 198.078,Z 396.072,A -85,B 0,C 180,E1 -21340.218,E2 -21340.218} C_VEL
LIN {X 0,Y 198.76,Z 394.959,A -85,B 0,C 180,E1 -21342.248,E2 -21342.248} C_VEL
LIN {X 0,Y 199.648,Z 393.413,A -85,B 0,C 180,E1 -21344.265,E2 -21344.265} C_VEL
LIN {X 0,Y 201.473,Z 390.327,A -85,B 0,C 180,E1 -21347.247,E2 -21347.247} C_VEL
LIN {X 0,Y 204.001,Z 386.206,A -85,B 0,C 180,E1 -21350.151,E2 -21350.151} C_VEL
LIN {X 0,Y 206.853,Z 380.967,A -85,B 0,C 180,E1 -21352.999,E2 -21352.999} C_VEL
LIN {X 0,Y 210.144,Z 374.483,A -85,B 0,C 180,E1 -21355.77,E2 -21355.77} C_VEL
LIN {X 0,Y 214.161,Z 366.473,A -85,B 0,C 180,E1 -21358.413,E2 -21358.413} C_VEL
LIN {X 0,Y 217.875,Z 358.369,A -85,B 0,C 180,E1 -21360.533,E2 -21360.533} C_VEL
LIN {X 0,Y 221.951,Z 348.567,A -85,B 0,C 180,E1 -21362.567,E2 -21362.567} C_VEL
LIN {X 0,Y 225.787,Z 337.694,A -85,B 0,C 180,E1 -21364.344,E2 -21364.344} C_VEL
LIN {X 0,Y 229.553,Z 325.526,A -85,B 0,C 180,E1 -21365.84,E2 -21365.84} C_VEL
LIN {X 0,Y 232.746,Z 312.73,A -85,B 0,C 180,E1 -21367.015,E2 -21367.015} C_VEL
LIN {X 0,Y 235.34,Z 298.722,A -85,B 0,C 180,E1 -21367.912,E2 -21367.912} C_VEL
LIN {X 0,Y 236.932,Z 285.374,A -85,B 0,C 180,E1 -21368.464,E2 -21368.464} C_VEL
LIN {X 0,Y 240.094,Z 246.167,A -85,B 0,C 180,E1 -21369.855,E2 -21369.855} C_VEL
LIN {X 0,Y 239.531,Z 243.877,A -85,B 0,C 180,E1 -21370.167,E2 -21370.167} C_VEL
LIN {X 0,Y 235.583,Z 234.041,A -85,B 0,C 180,E1 -21372.11,E2 -21372.11} C_VEL
LIN {X 0,Y 231.745,Z 225.989,A -85,B 0,C 180,E1 -21374.109,E2 -21374.109} C_VEL
LIN {X 0,Y 227.564,Z 218.09,A -85,B 0,C 180,E1 -21376.539,E2 -21376.539} C_VEL
LIN {X 0,Y 224.169,Z 212.466,A -85,B 0,C 180,E1 -21378.726,E2 -21378.726} C_VEL
LIN {X 0,Y 220.96,Z 207.351,A -85,B 0,C 180,E1 -21381.123,E2 -21381.123} C_VEL
LIN {X 0,Y 217.386,Z 201.682,A -85,B 0,C 180,E1 -21384.412,E2 -21384.412} C_VEL
LIN {X 0,Y 213.021,Z 195.608,A -85,B 0,C 180,E1 -21390.337,E2 -21390.337} C_VEL
LIN {X 0,Y 211.949,Z 194.02,A -85,B 0,C 180,E1 -21392.995,E2 -21392.995} C_VEL
LIN {X 0,Y 211.319,Z 193.201,A -85,B 0,C 180,E1 -21396.478,E2 -21396.478} C_VEL
LIN {X 0,Y 212.268,Z 193.47,A -85,B 0,C 180,E1 -21402.076,E2 -21402.076} C_VEL
LIN {X 0,Y 213.604,Z 195.262,A -85,B 0,C 180,E1 -21404.982,E2 -21404.982} C_VEL
LIN {X 0,Y 217.558,Z 199.348,A -85,B 0,C 180,E1 -21409.913,E2 -21409.913} C_VEL
LIN {X 0,Y 221.481,Z 204.718,A -85,B 0,C 180,E1 -21413.423,E2 -21413.423} C_VEL
LIN {X 0,Y 225.223,Z 209.722,A -85,B 0,C 180,E1 -21416.085,E2 -21416.085} C_VEL
LIN {X 0,Y 227.803,Z 213.756,A -85,B 0,C 180,E1 -21417.71,E2 -21417.71} C_VEL
LIN {X 0,Y 233.772,Z 224.1,A -85,B 0,C 180,E1 -21421.035,E2 -21421.035} C_VEL
LIN {X 0,Y 238.556,Z 234.098,A -85,B 0,C 180,E1 -21423.418,E2 -21423.418} C_VEL
LIN {X 0,Y 240.647,Z 239.042,A -85,B 0,C 180,E1 -21424.383,E2 -21424.383} C_VEL
LIN {X 0,Y 236.474,Z 286.211,A -85,B 0,C 180,E1 -21426.043,E2 -21426.043} C_VEL
LIN {X 0,Y 234.521,Z 299.067,A -85,B 0,C 180,E1 -21426.778,E2 -21426.778} C_VEL
LIN {X 0,Y 232.127,Z 310.791,A -85,B 0,C 180,E1 -21427.742,E2 -21427.742} C_VEL
LIN {X 0,Y 229.101,Z 322.495,A -85,B 0,C 180,E1 -21429.048,E2 -21429.048} C_VEL
LIN {X 0,Y 225.231,Z 334.582,A -85,B 0,C 180,E1 -21430.79,E2 -21430.79} C_VEL
LIN {X 0,Y 221.674,Z 344.211,A -85,B 0,C 180,E1 -21432.584,E2 -21432.584} C_VEL
LIN {X 0,Y 217.874,Z 352.947,A -85,B 0,C 180,E1 -21434.603,E2 -21434.603} C_VEL
LIN {X 0,Y 213.688,Z 361.736,A -85,B 0,C 180,E1 -21437.217,E2 -21437.217} C_VEL
LIN {X 0,Y 209.659,Z 369.424,A -85,B 0,C 180,E1 -21440.187,E2 -21440.187} C_VEL
LIN {X 0,Y 206.289,Z 375.167,A -85,B 0,C 180,E1 -21443.098,E2 -21443.098} C_VEL
LIN {X 0,Y 203.016,Z 380.447,A -85,B 0,C 180,E1 -21446.745,E2 -21446.745} C_VEL
LIN {X 0,Y 201.201,Z 383.075,A -85,B 0,C 180,E1 -21449.275,E2 -21449.275} C_VEL
LIN {X 0,Y 199.522,Z 385.261,A -85,B 0,C 180,E1 -21452.289,E2 -21452.289} C_VEL
LIN {X 0,Y 198.257,Z 386.534,A -85,B 0,C 180,E1 -21455.382,E2 -21455.382} C_VEL
LIN {X 0,Y 197.413,Z 386.883,A -85,B 0,C 180,E1 -21458.446,E2 -21458.446} C_VEL
LIN {X 0,Y 196.957,Z 386.328,A -85,B 0,C 180,E1 -21461.468,E2 -21461.468} C_VEL
LIN {X 0,Y 196.865,Z 384.153,A -85,B 0,C 180,E1 -21465.559,E2 -21465.559} C_VEL
LIN {X 0,Y 197.153,Z 381.591,A -85,B 0,C 180,E1 -21468.467,E2 -21468.467} C_VEL
LIN {X 0,Y 197.818,Z 376.934,A -85,B 0,C 180,E1 -21472.175,E2 -21472.175} C_VEL
LIN {X 0,Y 198.73,Z 371.216,A -85,B 0,C 180,E1 -21475.541,E2 -21475.541} C_VEL
LIN {X 0,Y 200.021,Z 364.019,A -85,B 0,C 180,E1 -21478.785,E2 -21478.785} C_VEL
LIN {X 0,Y 201.431,Z 356.745,A -85,B 0,C 180,E1 -21481.41,E2 -21481.41} C_VEL
LIN {X 0,Y 203.214,Z 347.715,A -85,B 0,C 180,E1 -21484.05,E2 -21484.05} C_VEL
LIN {X 0,Y 205.185,Z 337.267,A -85,B 0,C 180,E1 -21486.479,E2 -21486.479} C_VEL
LIN {X 0,Y 207.266,Z 325.509,A -85,B 0,C 180,E1 -21488.624,E2 -21488.624} C_VEL
LIN {X 0,Y 209.083,Z 313.187,A -85,B 0,C 180,E1 -21490.359,E2 -21490.359} C_VEL
LIN {X 0,Y 210.599,Z 301.014,A -85,B 0,C 180,E1 -21491.643,E2 -21491.643} C_VEL
LIN {X 0,Y 211.797,Z 288.122,A -85,B 0,C 180,E1 -21492.624,E2 -21492.624} C_VEL
LIN {X 0,Y 212.692,Z 272.769,A -85,B 0,C 180,E1 -21493.339,E2 -21493.339} C_VEL
LIN {X 0,Y 215.306,Z 218.916,A -85,B 0,C 180,E1 -21495.378,E2 -21495.378} C_VEL
LIN {X 0,Y 206.826,Z 194.723,A -85,B 0,C 180,E1 -21497.436,E2 -21497.436} C_VEL
LIN {X 0,Y 200.046,Z 179.272,A -85,B 0,C 180,E1 -21499.045,E2 -21499.045} C_VEL
LIN {X 0,Y 199.931,Z 178.582,A -85,B 0,C 180,E1 -21499.109,E2 -21499.109} C_VEL
LIN {X 0,Y 200.064,Z 178.562,A -85,B 0,C 180,E1 -21501.923,E2 -21501.923} C_VEL
LIN {X 0,Y 200.283,Z 178.54,A -85,B 0,C 180,E1 -21507.989,E2 -21507.989} C_VEL
LIN {X 0,Y 200.444,Z 178.521,A -85,B 0,C 180,E1 -21510,E2 -21510} C_VEL
LIN {X 0,Y 199.981,Z 178.579,A -85,B 0,C 180,E1 -21514.031,E2 -21514.031} C_VEL
LIN {X 0,Y 200.072,Z 178.568,A -85,B 0,C 180,E1 -21518.078,E2 -21518.078} C_VEL
LIN {X 0,Y 199.85,Z 178.592,A -85,B 0,C 180,E1 -21522.181,E2 -21522.181} C_VEL
LIN {X 0,Y 199.74,Z 178.602,A -85,B 0,C 180,E1 -21526.349,E2 -21526.349} C_VEL
LIN {X 0,Y 199.639,Z 178.614,A -85,B 0,C 180,E1 -21530.612,E2 -21530.612} C_VEL
LIN {X 0,Y 199.617,Z 178.618,A -85,B 0,C 180,E1 -21534.992,E2 -21534.992} C_VEL
LIN {X 0,Y 199.604,Z 178.618,A -85,B 0,C 180,E1 -21539.534,E2 -21539.534} C_VEL
LIN {X 0,Y 199.662,Z 178.603,A -85,B 0,C 180,E1 -21542.353,E2 -21542.353} C_VEL
LIN {X 0,Y 199.614,Z 178.619,A -85,B 0,C 180,E1 -21546.765,E2 -21546.765} C_VEL
LIN {X 0,Y 199.591,Z 178.62,A -85,B 0,C 180,E1 -21549.332,E2 -21549.332} C_VEL
LIN {X 0,Y 199.562,Z 178.615,A -85,B 0,C 180,E1 -21552.308,E2 -21552.308} C_VEL
LIN {X 0,Y 199.572,Z 178.616,A -85,B 0,C 180,E1 -21555.228,E2 -21555.228} C_VEL
LIN {X 0,Y 199.566,Z 178.623,A -85,B 0,C 180,E1 -21558.003,E2 -21558.003} C_VEL
LIN {X 0,Y 199.593,Z 178.623,A -85,B 0,C 180,E1 -21560.773,E2 -21560.773} C_VEL
LIN {X 0,Y 199.607,Z 178.605,A -85,B 0,C 180,E1 -21565.713,E2 -21565.713} C_VEL
LIN {X 0,Y 199.683,Z 178.596,A -85,B 0,C 180,E1 -21568.135,E2 -21568.135} C_VEL
LIN {X 0,Y 199.631,Z 178.619,A -85,B 0,C 180,E1 -21572.765,E2 -21572.765} C_VEL
LIN {X 0,Y 199.656,Z 178.609,A -85,B 0,C 180,E1 -21577.22,E2 -21577.22} C_VEL
LIN {X 0,Y 199.743,Z 178.582,A -85,B 0,C 180,E1 -21581.804,E2 -21581.804} C_VEL
LIN {X 0,Y 199.766,Z 178.594,A -85,B 0,C 180,E1 -21585.744,E2 -21585.744} C_VEL
LIN {X 0,Y 200.021,Z 178.567,A -85,B 0,C 180,E1 -21589.883,E2 -21589.883} C_VEL
LIN {X 0,Y 199.991,Z 178.559,A -85,B 0,C 180,E1 -21593.949,E2 -21593.949} C_VEL
LIN {X 0,Y 200.279,Z 178.529,A -85,B 0,C 180,E1 -21597.99,E2 -21597.99} C_VEL
LIN {X 0,Y 200.444,Z 178.515,A -85,B 0,C 180,E1 -21600.001,E2 -21600.001} C_VEL
LIN {X 0,Y 199.978,Z 178.57,A -85,B 0,C 180,E1 -21604.031,E2 -21604.031} C_VEL
LIN {X 0,Y 200.063,Z 178.555,A -85,B 0,C 180,E1 -21608.079,E2 -21608.079} C_VEL
LIN {X 0,Y 199.851,Z 178.59,A -85,B 0,C 180,E1 -21612.182,E2 -21612.182} C_VEL
LIN {X 0,Y 199.741,Z 178.595,A -85,B 0,C 180,E1 -21616.35,E2 -21616.35} C_VEL
LIN {X 0,Y 199.64,Z 178.616,A -85,B 0,C 180,E1 -21620.613,E2 -21620.613} C_VEL
LIN {X 0,Y 199.616,Z 178.615,A -85,B 0,C 180,E1 -21624.993,E2 -21624.993} C_VEL
LIN {X 0,Y 199.603,Z 178.621,A -85,B 0,C 180,E1 -21629.535,E2 -21629.535} C_VEL
LIN {X 0,Y 199.665,Z 178.603,A -85,B 0,C 180,E1 -21632.353,E2 -21632.353} C_VEL
LIN {X 0,Y 199.618,Z 178.617,A -85,B 0,C 180,E1 -21636.765,E2 -21636.765} C_VEL
LIN {X 0,Y 199.595,Z 178.621,A -85,B 0,C 180,E1 -21639.332,E2 -21639.332} C_VEL
LIN {X 0,Y 199.566,Z 178.626,A -85,B 0,C 180,E1 -21642.308,E2 -21642.308} C_VEL
LIN {X 0,Y 199.577,Z 178.625,A -85,B 0,C 180,E1 -21645.228,E2 -21645.228} C_VEL
LIN {X 0,Y 199.571,Z 178.625,A -85,B 0,C 180,E1 -21648.003,E2 -21648.003} C_VEL
LIN {X 0,Y 199.658,Z 178.804,A -85,B 0,C 180,E1 -21651.532,E2 -21651.532} C_VEL
LIN {X 0,Y 201.206,Z 185.796,A -85,B 0,C 180,E1 -21654.945,E2 -21654.945} C_VEL
LIN {X 0,Y 209.787,Z 209.28,A -85,B 0,C 180,E1 -21657.109,E2 -21657.109} C_VEL
LIN {X 0,Y 211.875,Z 216.226,A -85,B 0,C 180,E1 -21657.658,E2 -21657.658} C_VEL
LIN {X 0,Y 212.833,Z 223.454,A -85,B 0,C 180,E1 -21658.082,E2 -21658.082} C_VEL
LIN {X 0,Y 212.837,Z 229.283,A -85,B 0,C 180,E1 -21658.337,E2 -21658.337} C_VEL
LIN {X 0,Y 211.751,Z 235.123,A -85,B 0,C 180,E1 -21658.474,E2 -21658.474} C_VEL
LIN {X 0,Y 208.504,Z 246.746,A -85,B 0,C 180,E1 -21658.633,E2 -21658.633} C_VEL
LIN {X 0,Y 207.435,Z 252.653,A -85,B 0,C 180,E1 -21658.78,E2 -21658.78} C_VEL
LIN {X 0,Y 207.304,Z 254.639,A -85,B 0,C 180,E1 -21658.855,E2 -21658.855} C_VEL
LIN {X 0,Y 205.268,Z 294.092,A -85,B 0,C 180,E1 -21660.446,E2 -21660.446} C_VEL
LIN {X 0,Y 204.048,Z 307.953,A -85,B 0,C 180,E1 -21661.382,E2 -21661.382} C_VEL
LIN {X 0,Y 202.473,Z 320.562,A -85,B 0,C 180,E1 -21662.618,E2 -21662.618} C_VEL
LIN {X 0,Y 200.336,Z 332.979,A -85,B 0,C 180,E1 -21664.27,E2 -21664.27} C_VEL
LIN {X 0,Y 198.303,Z 344.232,A -85,B 0,C 180,E1 -21666.225,E2 -21666.225} C_VEL
LIN {X 0,Y 196.524,Z 353.647,A -85,B 0,C 180,E1 -21668.284,E2 -21668.284} C_VEL
LIN {X 0,Y 194.955,Z 361.987,A -85,B 0,C 180,E1 -21670.521,E2 -21670.521} C_VEL
LIN {X 0,Y 193.134,Z 371.252,A -85,B 0,C 180,E1 -21673.619,E2 -21673.619} C_VEL
LIN {X 0,Y 191.7,Z 378.683,A -85,B 0,C 180,E1 -21676.754,E2 -21676.754} C_VEL
LIN {X 0,Y 190.949,Z 383.693,A -85,B 0,C 180,E1 -21679.395,E2 -21679.395} C_VEL
LIN {X 0,Y 190.44,Z 388.524,A -85,B 0,C 180,E1 -21682.578,E2 -21682.578} C_VEL
LIN {X 0,Y 190.192,Z 392.537,A -85,B 0,C 180,E1 -21686.132,E2 -21686.132} C_VEL
LIN {X 0,Y 190.228,Z 394.016,A -85,B 0,C 180,E1 -21687.882,E2 -21687.882} C_VEL
LIN {X 0,Y 190.351,Z 395.379,A -85,B 0,C 180,E1 -21690,E2 -21690} C_VEL
LIN {X 0,Y 190.163,Z 396.745,A -85,B 0,C 180,E1 -21693.738,E2 -21693.738} C_VEL
LIN {X 0,Y 190.283,Z 396.98,A -85,B 0,C 180,E1 -21696.361,E2 -21696.361} C_VEL
LIN {X 0,Y 191.072,Z 396.021,A -85,B 0,C 180,E1 -21700.597,E2 -21700.597} C_VEL
LIN {X 0,Y 192.741,Z 393.526,A -85,B 0,C 180,E1 -21704.787,E2 -21704.787} C_VEL
LIN {X 0,Y 194.707,Z 390.538,A -85,B 0,C 180,E1 -21707.866,E2 -21707.866} C_VEL
LIN {X 0,Y 197.36,Z 386.559,A -85,B 0,C 180,E1 -21710.86,E2 -21710.86} C_VEL
LIN {X 0,Y 200.349,Z 381.509,A -85,B 0,C 180,E1 -21713.791,E2 -21713.791} C_VEL
LIN {X 0,Y 203.825,Z 375.236,A -85,B 0,C 180,E1 -21716.63,E2 -21716.63} C_VEL
LIN {X 0,Y 208.009,Z 367.44,A -85,B 0,C 180,E1 -21719.334,E2 -21719.334} C_VEL
LIN {X 0,Y 211.874,Z 359.556,A -85,B 0,C 180,E1 -21721.495,E2 -21721.495} C_VEL
LIN {X 0,Y 216.532,Z 349.035,A -85,B 0,C 180,E1 -21723.767,E2 -21723.767} C_VEL
LIN {X 0,Y 220.56,Z 338.449,A -85,B 0,C 180,E1 -21725.557,E2 -21725.557} C_VEL
LIN {X 0,Y 224.459,Z 326.566,A -85,B 0,C 180,E1 -21727.065,E2 -21727.065} C_VEL
LIN {X 0,Y 227.772,Z 314.192,A -85,B 0,C 180,E1 -21728.245,E2 -21728.245} C_VEL
LIN {X 0,Y 230.411,Z 301.236,A -85,B 0,C 180,E1 -21729.124,E2 -21729.124} C_VEL
LIN {X 0,Y 232.275,Z 287.523,A -85,B 0,C 180,E1 -21729.743,E2 -21729.743} C_VEL
LIN {X 0,Y 235.644,Z 248.225,A -85,B 0,C 180,E1 -21731.145,E2 -21731.145} C_VEL
LIN {X 0,Y 232.112,Z 238.946,A -85,B 0,C 180,E1 -21733.042,E2 -21733.042} C_VEL
LIN {X 0,Y 228.627,Z 231.304,A -85,B 0,C 180,E1 -21734.992,E2 -21734.992} C_VEL
LIN {X 0,Y 224.743,Z 223.701,A -85,B 0,C 180,E1 -21737.404,E2 -21737.404} C_VEL
LIN {X 0,Y 221.827,Z 218.573,A -85,B 0,C 180,E1 -21739.442,E2 -21739.442} C_VEL
LIN {X 0,Y 218.888,Z 213.673,A -85,B 0,C 180,E1 -21741.763,E2 -21741.763} C_VEL
LIN {X 0,Y 215.515,Z 208.133,A -85,B 0,C 180,E1 -21745.093,E2 -21745.093} C_VEL
LIN {X 0,Y 211.738,Z 202.52,A -85,B 0,C 180,E1 -21750.65,E2 -21750.65} C_VEL
LIN {X 0,Y 210.742,Z 200.934,A -85,B 0,C 180,E1 -21753.262,E2 -21753.262} C_VEL
LIN {X 0,Y 210.218,Z 200.233,A -85,B 0,C 180,E1 -21756.347,E2 -21756.347} C_VEL
LIN {X 0,Y 210.969,Z 200.366,A -85,B 0,C 180,E1 -21761.607,E2 -21761.607} C_VEL
LIN {X 0,Y 212.097,Z 201.788,A -85,B 0,C 180,E1 -21764.258,E2 -21764.258} C_VEL
LIN {X 0,Y 215.871,Z 205.984,A -85,B 0,C 180,E1 -21769.412,E2 -21769.412} C_VEL
LIN {X 0,Y 219.542,Z 211.296,A -85,B 0,C 180,E1 -21772.91,E2 -21772.91} C_VEL
LIN {X 0,Y 222.959,Z 215.972,A -85,B 0,C 180,E1 -21775.442,E2 -21775.442} C_VEL
LIN {X 0,Y 225.205,Z 219.708,A -85,B 0,C 180,E1 -21776.978,E2 -21776.978} C_VEL
LIN {X 0,Y 230.875,Z 229.962,A -85,B 0,C 180,E1 -21780.34,E2 -21780.34} C_VEL
LIN {X 0,Y 235.464,Z 240.121,A -85,B 0,C 180,E1 -21782.753,E2 -21782.753} C_VEL
LIN {X 0,Y 236.156,Z 241.813,A -85,B 0,C 180,E1 -21783.107,E2 -21783.107} C_VEL
LIN {X 0,Y 232.036,Z 286.004,A -85,B 0,C 180,E1 -21784.667,E2 -21784.667} C_VEL
LIN {X 0,Y 229.861,Z 299.943,A -85,B 0,C 180,E1 -21785.478,E2 -21785.478} C_VEL
LIN {X 0,Y 227.146,Z 312.377,A -85,B 0,C 180,E1 -21786.539,E2 -21786.539} C_VEL
LIN {X 0,Y 223.883,Z 324.131,A -85,B 0,C 180,E1 -21787.893,E2 -21787.893} C_VEL
LIN {X 0,Y 220.443,Z 334.261,A -85,B 0,C 180,E1 -21789.379,E2 -21789.379} C_VEL
LIN {X 0,Y 216.548,Z 344.19,A -85,B 0,C 180,E1 -21791.228,E2 -21791.228} C_VEL
LIN {X 0,Y 212.372,Z 353.351,A -85,B 0,C 180,E1 -21793.393,E2 -21793.393} C_VEL
LIN {X 0,Y 207.962,Z 362.109,A -85,B 0,C 180,E1 -21796.046,E2 -21796.046} C_VEL
LIN {X 0,Y 203.646,Z 369.785,A -85,B 0,C 180,E1 -21799.076,E2 -21799.076} C_VEL
LIN {X 0,Y 199.907,Z 375.73,A -85,B 0,C 180,E1 -21802.205,E2 -21802.205} C_VEL
LIN {X 0,Y 196.936,Z 380.178,A -85,B 0,C 180,E1 -21805.355,E2 -21805.355} C_VEL
LIN {X 0,Y 194.91,Z 382.936,A -85,B 0,C 180,E1 -21807.952,E2 -21807.952} C_VEL
LIN {X 0,Y 193.252,Z 384.965,A -85,B 0,C 180,E1 -21810.605,E2 -21810.605} C_VEL
LIN {X 0,Y 191.922,Z 386.315,A -85,B 0,C 180,E1 -21813.317,E2 -21813.317} C_VEL
LIN {X 0,Y 190.914,Z 387.019,A -85,B 0,C 180,E1 -21816.085,E2 -21816.085} C_VEL
LIN {X 0,Y 190.173,Z 386.965,A -85,B 0,C 180,E1 -21819.099,E2 -21819.099} C_VEL
LIN {X 0,Y 189.8,Z 386.065,A -85,B 0,C 180,E1 -21822.222,E2 -21822.222} C_VEL
LIN {X 0,Y 189.762,Z 384.342,A -85,B 0,C 180,E1 -21825.278,E2 -21825.278} C_VEL
LIN {X 0,Y 190.039,Z 381.806,A -85,B 0,C 180,E1 -21828.267,E2 -21828.267} C_VEL
LIN {X 0,Y 190.495,Z 378.481,A -85,B 0,C 180,E1 -21831.158,E2 -21831.158} C_VEL
LIN {X 0,Y 191.393,Z 373.103,A -85,B 0,C 180,E1 -21834.667,E2 -21834.667} C_VEL
LIN {X 0,Y 192.66,Z 365.808,A -85,B 0,C 180,E1 -21838.306,E2 -21838.306} C_VEL
LIN {X 0,Y 194.185,Z 358.205,A -85,B 0,C 180,E1 -21841.264,E2 -21841.264} C_VEL
LIN {X 0,Y 196.09,Z 348.767,A -85,B 0,C 180,E1 -21844.182,E2 -21844.182} C_VEL
LIN {X 0,Y 198.139,Z 338.28,A -85,B 0,C 180,E1 -21846.759,E2 -21846.759} C_VEL
LIN {X 0,Y 200.166,Z 327.104,A -85,B 0,C 180,E1 -21848.907,E2 -21848.907} C_VEL
LIN {X 0,Y 202.085,Z 314.922,A -85,B 0,C 180,E1 -21850.741,E2 -21850.741} C_VEL
LIN {X 0,Y 203.693,Z 302.824,A -85,B 0,C 180,E1 -21852.103,E2 -21852.103} C_VEL
LIN {X 0,Y 205.024,Z 289.136,A -85,B 0,C 180,E1 -21853.212,E2 -21853.212} C_VEL
LIN {X 0,Y 205.982,Z 275.032,A -85,B 0,C 180,E1 -21853.916,E2 -21853.916} C_VEL
LIN {X 0,Y 208.603,Z 220.197,A -85,B 0,C 180,E1 -21856.073,E2 -21856.073} C_VEL
LIN {X 0,Y 200.414,Z 196.72,A -85,B 0,C 180,E1 -21858.168,E2 -21858.168} C_VEL
LIN {X 0,Y 193.069,Z 180.038,A -85,B 0,C 180,E1 -21860.002,E2 -21860.002} C_VEL
LIN {X 0,Y 192.967,Z 179.45,A -85,B 0,C 180,E1 -21860.139,E2 -21860.139} C_VEL
LIN {X 0,Y 192.96,Z 179.449,A -85,B 0,C 180,E1 -21863.727,E2 -21863.727} C_VEL
LIN {X 0,Y 193.227,Z 179.418,A -85,B 0,C 180,E1 -21867.916,E2 -21867.916} C_VEL
LIN {X 0,Y 193.41,Z 179.397,A -85,B 0,C 180,E1 -21870,E2 -21870} C_VEL
LIN {X 0,Y 192.929,Z 179.457,A -85,B 0,C 180,E1 -21874.178,E2 -21874.178} C_VEL
LIN {X 0,Y 193.023,Z 179.444,A -85,B 0,C 180,E1 -21878.375,E2 -21878.375} C_VEL
LIN {X 0,Y 192.772,Z 179.473,A -85,B 0,C 180,E1 -21882.636,E2 -21882.636} C_VEL
LIN {X 0,Y 192.692,Z 179.482,A -85,B 0,C 180,E1 -21888.509,E2 -21888.509} C_VEL
LIN {X 0,Y 192.608,Z 179.49,A -85,B 0,C 180,E1 -21894.189,E2 -21894.189} C_VEL
LIN {X 0,Y 192.597,Z 179.493,A -85,B 0,C 180,E1 -21898.865,E2 -21898.865} C_VEL
LIN {X 0,Y 192.592,Z 179.485,A -85,B 0,C 180,E1 -21903.187,E2 -21903.187} C_VEL
LIN {X 0,Y 192.538,Z 179.5,A -85,B 0,C 180,E1 -21908.355,E2 -21908.355} C_VEL
LIN {X 0,Y 192.481,Z 179.493,A -85,B 0,C 180,E1 -21913.094,E2 -21913.094} C_VEL
LIN {X 0,Y 192.481,Z 179.504,A -85,B 0,C 180,E1 -21916.907,E2 -21916.907} C_VEL
LIN {X 0,Y 192.538,Z 179.498,A -85,B 0,C 180,E1 -21921.646,E2 -21921.646} C_VEL
LIN {X 0,Y 192.592,Z 179.476,A -85,B 0,C 180,E1 -21926.814,E2 -21926.814} C_VEL
LIN {X 0,Y 192.616,Z 179.488,A -85,B 0,C 180,E1 -21931.685,E2 -21931.685} C_VEL
LIN {X 0,Y 192.643,Z 179.487,A -85,B 0,C 180,E1 -21936.341,E2 -21936.341} C_VEL
LIN {X 0,Y 192.692,Z 179.459,A -85,B 0,C 180,E1 -21941.493,E2 -21941.493} C_VEL
LIN {X 0,Y 192.771,Z 179.468,A -85,B 0,C 180,E1 -21947.365,E2 -21947.365} C_VEL
LIN {X 0,Y 193.015,Z 179.436,A -85,B 0,C 180,E1 -21951.626,E2 -21951.626} C_VEL
LIN {X 0,Y 193.223,Z 179.407,A -85,B 0,C 180,E1 -21957.916,E2 -21957.916} C_VEL
LIN {X 0,Y 193.41,Z 179.391,A -85,B 0,C 180,E1 -21960.001,E2 -21960.001} C_VEL
LIN {X 0,Y 192.926,Z 179.447,A -85,B 0,C 180,E1 -21964.179,E2 -21964.179} C_VEL
LIN {X 0,Y 193.016,Z 179.435,A -85,B 0,C 180,E1 -21968.376,E2 -21968.376} C_VEL
LIN {X 0,Y 192.773,Z 179.471,A -85,B 0,C 180,E1 -21972.636,E2 -21972.636} C_VEL
LIN {X 0,Y 192.694,Z 179.479,A -85,B 0,C 180,E1 -21978.509,E2 -21978.509} C_VEL
LIN {X 0,Y 192.609,Z 179.487,A -85,B 0,C 180,E1 -21984.188,E2 -21984.188} C_VEL
LIN {X 0,Y 192.594,Z 179.496,A -85,B 0,C 180,E1 -21988.862,E2 -21988.862} C_VEL
LIN {X 0,Y 192.595,Z 179.478,A -85,B 0,C 180,E1 -21993.188,E2 -21993.188} C_VEL
LIN {X 0,Y 192.542,Z 179.5,A -85,B 0,C 180,E1 -21998.355,E2 -21998.355} C_VEL
LIN {X 0,Y 192.485,Z 179.509,A -85,B 0,C 180,E1 -22003.094,E2 -22003.094} C_VEL
LIN {X 0,Y 192.486,Z 179.509,A -85,B 0,C 180,E1 -22006.907,E2 -22006.907} C_VEL
LIN {X 0,Y 192.574,Z 179.6,A -85,B 0,C 180,E1 -22010.868,E2 -22010.868} C_VEL
LIN {X 0,Y 193.939,Z 185.513,A -85,B 0,C 180,E1 -22013.904,E2 -22013.904} C_VEL
LIN {X 0,Y 201.416,Z 205.549,A -85,B 0,C 180,E1 -22015.909,E2 -22015.909} C_VEL
LIN {X 0,Y 205.384,Z 217.581,A -85,B 0,C 180,E1 -22016.962,E2 -22016.962} C_VEL
LIN {X 0,Y 208.021,Z 239.587,A -85,B 0,C 180,E1 -22018.263,E2 -22018.263} C_VEL
LIN {X 0,Y 207.304,Z 254.639,A -85,B 0,C 180,E1 -22018.855,E2 -22018.855} C_VEL
LIN {X 0,Y 206.479,Z 260.445,A -85,B 0,C 180,E1 -22019.026,E2 -22019.026} C_VEL
LIN {X 0,Y 200.17,Z 279.245,A -85,B 0,C 180,E1 -22019.196,E2 -22019.196} C_VEL
LIN {X 0,Y 199.217,Z 285.056,A -85,B 0,C 180,E1 -22019.362,E2 -22019.362} C_VEL
LIN {X 0,Y 198.175,Z 299.456,A -85,B 0,C 180,E1 -22020.086,E2 -22020.086} C_VEL
LIN {X 0,Y 196.684,Z 312.667,A -85,B 0,C 180,E1 -22021.159,E2 -22021.159} C_VEL
LIN {X 0,Y 194.929,Z 325.468,A -85,B 0,C 180,E1 -22022.633,E2 -22022.633} C_VEL
LIN {X 0,Y 192.914,Z 336.799,A -85,B 0,C 180,E1 -22024.366,E2 -22024.366} C_VEL
LIN {X 0,Y 190.843,Z 347.223,A -85,B 0,C 180,E1 -22026.392,E2 -22026.392} C_VEL
LIN {X 0,Y 188.587,Z 357.956,A -85,B 0,C 180,E1 -22029.029,E2 -22029.029} C_VEL
LIN {X 0,Y 187.123,Z 365.623,A -85,B 0,C 180,E1 -22031.383,E2 -22031.383} C_VEL
LIN {X 0,Y 185.413,Z 374.112,A -85,B 0,C 180,E1 -22034.613,E2 -22034.613} C_VEL
LIN {X 0,Y 184.241,Z 380.931,A -85,B 0,C 180,E1 -22037.889,E2 -22037.889} C_VEL
LIN {X 0,Y 183.539,Z 386.333,A -85,B 0,C 180,E1 -22041.189,E2 -22041.189} C_VEL
LIN {X 0,Y 183.199,Z 390.48,A -85,B 0,C 180,E1 -22044.496,E2 -22044.496} C_VEL
LIN {X 0,Y 183.136,Z 393.509,A -85,B 0,C 180,E1 -22047.8,E2 -22047.8} C_VEL
LIN {X 0,Y 183.271,Z 394.974,A -85,B 0,C 180,E1 -22050,E2 -22050} C_VEL
LIN {X 0,Y 183.077,Z 396.385,A -85,B 0,C 180,E1 -22053.522,E2 -22053.522} C_VEL
LIN {X 0,Y 183.216,Z 396.76,A -85,B 0,C 180,E1 -22056.608,E2 -22056.608} C_VEL
LIN {X 0,Y 183.525,Z 396.576,A -85,B 0,C 180,E1 -22058.811,E2 -22058.811} C_VEL
LIN {X 0,Y 184.854,Z 394.975,A -85,B 0,C 180,E1 -22063.186,E2 -22063.186} C_VEL
LIN {X 0,Y 187.154,Z 391.842,A -85,B 0,C 180,E1 -22067.482,E2 -22067.482} C_VEL
LIN {X 0,Y 189.741,Z 388.345,A -85,B 0,C 180,E1 -22070.602,E2 -22070.602} C_VEL
LIN {X 0,Y 192.877,Z 383.806,A -85,B 0,C 180,E1 -22073.628,E2 -22073.628} C_VEL
LIN {X 0,Y 196.237,Z 378.137,A -85,B 0,C 180,E1 -22076.592,E2 -22076.592} C_VEL
LIN {X 0,Y 200.483,Z 371.096,A -85,B 0,C 180,E1 -22079.391,E2 -22079.391} C_VEL
LIN {X 0,Y 203.419,Z 365.544,A -85,B 0,C 180,E1 -22081.213,E2 -22081.213} C_VEL
LIN {X 0,Y 207.698,Z 357.365,A -85,B 0,C 180,E1 -22083.357,E2 -22083.357} C_VEL
LIN {X 0,Y 212.156,Z 347.507,A -85,B 0,C 180,E1 -22085.429,E2 -22085.429} C_VEL
LIN {X 0,Y 216.436,Z 336.514,A -85,B 0,C 180,E1 -22087.212,E2 -22087.212} C_VEL
LIN {X 0,Y 220.028,Z 325.906,A -85,B 0,C 180,E1 -22088.524,E2 -22088.524} C_VEL
LIN {X 0,Y 223.454,Z 313.478,A -85,B 0,C 180,E1 -22089.706,E2 -22089.706} C_VEL
LIN {X 0,Y 226.176,Z 300.422,A -85,B 0,C 180,E1 -22090.585,E2 -22090.585} C_VEL
LIN {X 0,Y 228.133,Z 286.576,A -85,B 0,C 180,E1 -22091.196,E2 -22091.196} C_VEL
LIN {X 0,Y 231.358,Z 250.834,A -85,B 0,C 180,E1 -22092.492,E2 -22092.492} C_VEL
LIN {X 0,Y 227.41,Z 240.616,A -85,B 0,C 180,E1 -22094.786,E2 -22094.786} C_VEL
LIN {X 0,Y 223.76,Z 232.86,A -85,B 0,C 180,E1 -22097.086,E2 -22097.086} C_VEL
LIN {X 0,Y 221.537,Z 228.496,A -85,B 0,C 180,E1 -22098.63,E2 -22098.63} C_VEL
LIN {X 0,Y 219.353,Z 224.418,A -85,B 0,C 180,E1 -22100.303,E2 -22100.303} C_VEL
LIN {X 0,Y 216.862,Z 220.023,A -85,B 0,C 180,E1 -22102.439,E2 -22102.439} C_VEL
LIN {X 0,Y 213.727,Z 214.629,A -85,B 0,C 180,E1 -22105.744,E2 -22105.744} C_VEL
LIN {X 0,Y 210.354,Z 209.189,A -85,B 0,C 180,E1 -22111.232,E2 -22111.232} C_VEL
LIN {X 0,Y 209.52,Z 207.853,A -85,B 0,C 180,E1 -22113.651,E2 -22113.651} C_VEL
LIN {X 0,Y 209.141,Z 207.129,A -85,B 0,C 180,E1 -22118.305,E2 -22118.305} C_VEL
LIN {X 0,Y 210.202,Z 207.677,A -85,B 0,C 180,E1 -22122.487,E2 -22122.487} C_VEL
LIN {X 0,Y 214.249,Z 212.726,A -85,B 0,C 180,E1 -22128.957,E2 -22128.957} C_VEL
LIN {X 0,Y 217.614,Z 217.787,A -85,B 0,C 180,E1 -22132.33,E2 -22132.33} C_VEL
LIN {X 0,Y 220.844,Z 222.415,A -85,B 0,C 180,E1 -22134.874,E2 -22134.874} C_VEL
LIN {X 0,Y 223.146,Z 226.608,A -85,B 0,C 180,E1 -22136.561,E2 -22136.561} C_VEL
LIN {X 0,Y 227.91,Z 235.559,A -85,B 0,C 180,E1 -22139.53,E2 -22139.53} C_VEL
LIN {X 0,Y 231.889,Z 244.776,A -85,B 0,C 180,E1 -22141.782,E2 -22141.782} C_VEL
LIN {X 0,Y 227.774,Z 286.344,A -85,B 0,C 180,E1 -22143.255,E2 -22143.255} C_VEL
LIN {X 0,Y 225.462,Z 300.355,A -85,B 0,C 180,E1 -22144.079,E2 -22144.079} C_VEL
LIN {X 0,Y 222.849,Z 311.772,A -85,B 0,C 180,E1 -22145.044,E2 -22145.044} C_VEL
LIN {X 0,Y 219.261,Z 324.173,A -85,B 0,C 180,E1 -22146.472,E2 -22146.472} C_VEL
LIN {X 0,Y 215.21,Z 335.588,A -85,B 0,C 180,E1 -22148.172,E2 -22148.172} C_VEL
LIN {X 0,Y 211.081,Z 345.409,A -85,B 0,C 180,E1 -22150.066,E2 -22150.066} C_VEL
LIN {X 0,Y 206.183,Z 355.44,A -85,B 0,C 180,E1 -22152.55,E2 -22152.55} C_VEL
LIN {X 0,Y 201.685,Z 363.687,A -85,B 0,C 180,E1 -22155.216,E2 -22155.216} C_VEL
LIN {X 0,Y 197.734,Z 370.139,A -85,B 0,C 180,E1 -22157.898,E2 -22157.898} C_VEL
LIN {X 0,Y 193.537,Z 376.367,A -85,B 0,C 180,E1 -22161.292,E2 -22161.292} C_VEL
LIN {X 0,Y 190.979,Z 379.953,A -85,B 0,C 180,E1 -22163.878,E2 -22163.878} C_VEL
LIN {X 0,Y 187.731,Z 383.944,A -85,B 0,C 180,E1 -22167.899,E2 -22167.899} C_VEL
LIN {X 0,Y 185.331,Z 386.38,A -85,B 0,C 180,E1 -22172.065,E2 -22172.065} C_VEL
LIN {X 0,Y 183.655,Z 387.289,A -85,B 0,C 180,E1 -22176.525,E2 -22176.525} C_VEL
LIN {X 0,Y 182.8,Z 386.639,A -85,B 0,C 180,E1 -22180.811,E2 -22180.811} C_VEL
LIN {X 0,Y 182.65,Z 385.242,A -85,B 0,C 180,E1 -22183.835,E2 -22183.835} C_VEL
LIN {X 0,Y 182.766,Z 382.996,A -85,B 0,C 180,E1 -22186.937,E2 -22186.937} C_VEL
LIN {X 0,Y 183.197,Z 379.791,A -85,B 0,C 180,E1 -22190.107,E2 -22190.107} C_VEL
LIN {X 0,Y 183.903,Z 375.417,A -85,B 0,C 180,E1 -22193.371,E2 -22193.371} C_VEL
LIN {X 0,Y 184.903,Z 369.599,A -85,B 0,C 180,E1 -22196.739,E2 -22196.739} C_VEL
LIN {X 0,Y 186.362,Z 362.082,A -85,B 0,C 180,E1 -22200.152,E2 -22200.152} C_VEL
LIN {X 0,Y 188.055,Z 353.976,A -85,B 0,C 180,E1 -22203.056,E2 -22203.056} C_VEL
LIN {X 0,Y 190.243,Z 343.569,A -85,B 0,C 180,E1 -22206.024,E2 -22206.024} C_VEL
LIN {X 0,Y 192.214,Z 333.521,A -85,B 0,C 180,E1 -22208.288,E2 -22208.288} C_VEL
LIN {X 0,Y 194.297,Z 321.756,A -85,B 0,C 180,E1 -22210.375,E2 -22210.375} C_VEL
LIN {X 0,Y 196.073,Z 310.014,A -85,B 0,C 180,E1 -22211.992,E2 -22211.992} C_VEL
LIN {X 0,Y 197.584,Z 297.14,A -85,B 0,C 180,E1 -22213.302,E2 -22213.302} C_VEL
LIN {X 0,Y 198.823,Z 283.044,A -85,B 0,C 180,E1 -22214.277,E2 -22214.277} C_VEL
LIN {X 0,Y 202.103,Z 222.235,A -85,B 0,C 180,E1 -22216.757,E2 -22216.757} C_VEL
LIN {X 0,Y 195.378,Z 202.318,A -85,B 0,C 180,E1 -22218.583,E2 -22218.583} C_VEL
LIN {X 0,Y 188.275,Z 186.014,A -85,B 0,C 180,E1 -22220.398,E2 -22220.398} C_VEL
LIN {X 0,Y 186.115,Z 181.229,A -85,B 0,C 180,E1 -22220.971,E2 -22220.971} C_VEL
LIN {X 0,Y 185.951,Z 180.319,A -85,B 0,C 180,E1 -22221.1,E2 -22221.1} C_VEL
LIN {X 0,Y 186.173,Z 180.297,A -85,B 0,C 180,E1 -22227.837,E2 -22227.837} C_VEL
LIN {X 0,Y 186.376,Z 180.273,A -85,B 0,C 180,E1 -22230,E2 -22230} C_VEL
LIN {X 0,Y 185.878,Z 180.336,A -85,B 0,C 180,E1 -22234.337,E2 -22234.337} C_VEL
LIN {X 0,Y 185.972,Z 180.322,A -85,B 0,C 180,E1 -22238.695,E2 -22238.695} C_VEL
LIN {X 0,Y 185.696,Z 180.355,A -85,B 0,C 180,E1 -22243.125,E2 -22243.125} C_VEL
LIN {X 0,Y 185.622,Z 180.363,A -85,B 0,C 180,E1 -22248.821,E2 -22248.821} C_VEL
LIN {X 0,Y 185.542,Z 180.37,A -85,B 0,C 180,E1 -22254.624,E2 -22254.624} C_VEL
LIN {X 0,Y 185.541,Z 180.369,A -85,B 0,C 180,E1 -22259.5,E2 -22259.5} C_VEL
LIN {X 0,Y 185.494,Z 180.374,A -85,B 0,C 180,E1 -22264.633,E2 -22264.633} C_VEL
LIN {X 0,Y 185.497,Z 180.38,A -85,B 0,C 180,E1 -22267.315,E2 -22267.315} C_VEL
LIN {X 0,Y 185.458,Z 180.378,A -85,B 0,C 180,E1 -22270.721,E2 -22270.721} C_VEL
LIN {X 0,Y 185.452,Z 180.377,A -85,B 0,C 180,E1 -22276.057,E2 -22276.057} C_VEL
LIN {X 0,Y 185.453,Z 180.382,A -85,B 0,C 180,E1 -22279.893,E2 -22279.893} C_VEL
LIN {X 0,Y 185.498,Z 180.374,A -85,B 0,C 180,E1 -22282.715,E2 -22282.715} C_VEL
LIN {X 0,Y 185.528,Z 180.358,A -85,B 0,C 180,E1 -22287.973,E2 -22287.973} C_VEL
LIN {X 0,Y 185.544,Z 180.366,A -85,B 0,C 180,E1 -22290.596,E2 -22290.596} C_VEL
LIN {X 0,Y 185.542,Z 180.371,A -85,B 0,C 180,E1 -22295.377,E2 -22295.377} C_VEL
LIN {X 0,Y 185.623,Z 180.339,A -85,B 0,C 180,E1 -22301.18,E2 -22301.18} C_VEL
LIN {X 0,Y 185.695,Z 180.35,A -85,B 0,C 180,E1 -22306.876,E2 -22306.876} C_VEL
LIN {X 0,Y 185.967,Z 180.313,A -85,B 0,C 180,E1 -22311.306,E2 -22311.306} C_VEL
LIN {X 0,Y 186.169,Z 180.285,A -85,B 0,C 180,E1 -22317.837,E2 -22317.837} C_VEL
LIN {X 0,Y 186.376,Z 180.267,A -85,B 0,C 180,E1 -22320.001,E2 -22320.001} C_VEL
LIN {X 0,Y 185.874,Z 180.325,A -85,B 0,C 180,E1 -22324.338,E2 -22324.338} C_VEL
LIN {X 0,Y 185.968,Z 180.313,A -85,B 0,C 180,E1 -22328.695,E2 -22328.695} C_VEL
LIN {X 0,Y 185.698,Z 180.353,A -85,B 0,C 180,E1 -22333.126,E2 -22333.126} C_VEL
LIN {X 0,Y 185.624,Z 180.36,A -85,B 0,C 180,E1 -22338.822,E2 -22338.822} C_VEL
LIN {X 0,Y 185.544,Z 180.366,A -85,B 0,C 180,E1 -22344.625,E2 -22344.625} C_VEL
LIN {X 0,Y 185.518,Z 180.376,A -85,B 0,C 180,E1 -22349.505,E2 -22349.505} C_VEL
LIN {X 0,Y 185.529,Z 180.357,A -85,B 0,C 180,E1 -22353.553,E2 -22353.553} C_VEL
LIN {X 0,Y 185.5,Z 180.379,A -85,B 0,C 180,E1 -22357.315,E2 -22357.315} C_VEL
LIN {X 0,Y 185.462,Z 180.382,A -85,B 0,C 180,E1 -22360.722,E2 -22360.722} C_VEL
LIN {X 0,Y 185.456,Z 180.383,A -85,B 0,C 180,E1 -22366.057,E2 -22366.057} C_VEL
